LIN {X 0,Y 485.408,Z 513.857,A -85,B 0,C 180,E1 -6732.652,E2 -6732.652} C_VEL
LIN {X 0,Y 484.952,Z 527.725,A -85,B 0,C 180,E1 -6733.189,E2 -6733.189} C_VEL
LIN {X 0,Y 484.519,Z 541.1,A -85,B 0,C 180,E1 -6733.893,E2 -6733.893} C_VEL
LIN {X 0,Y 483.878,Z 553.705,A -85,B 0,C 180,E1 -6734.736,E2 -6734.736} C_VEL
LIN {X 0,Y 483.305,Z 565.203,A -85,B 0,C 180,E1 -6735.687,E2 -6735.687} C_VEL
LIN {X 0,Y 482.695,Z 575.753,A -85,B 0,C 180,E1 -6736.742,E2 -6736.742} C_VEL
LIN {X 0,Y 482.294,Z 585.397,A -85,B 0,C 180,E1 -6737.906,E2 -6737.906} C_VEL
LIN {X 0,Y 481.754,Z 594.848,A -85,B 0,C 180,E1 -6739.28,E2 -6739.28} C_VEL
LIN {X 0,Y 481.429,Z 602.033,A -85,B 0,C 180,E1 -6740.547,E2 -6740.547} C_VEL
LIN {X 0,Y 481.163,Z 608.903,A -85,B 0,C 180,E1 -6742.023,E2 -6742.023} C_VEL
LIN {X 0,Y 481.013,Z 614.317,A -85,B 0,C 180,E1 -6743.484,E2 -6743.484} C_VEL
LIN {X 0,Y 480.898,Z 618.563,A -85,B 0,C 180,E1 -6744.968,E2 -6744.968} C_VEL
LIN {X 0,Y 480.881,Z 621.983,A -85,B 0,C 180,E1 -6746.648,E2 -6746.648} C_VEL
LIN {X 0,Y 480.789,Z 624.022,A -85,B 0,C 180,E1 -6748.324,E2 -6748.324} C_VEL
LIN {X 0,Y 480.742,Z 624.729,A -85,B 0,C 180,E1 -6749.999,E2 -6749.999} C_VEL
LIN {X 0,Y 480.787,Z 624.108,A -85,B 0,C 180,E1 -6751.674,E2 -6751.674} C_VEL
LIN {X 0,Y 480.88,Z 622.144,A -85,B 0,C 180,E1 -6753.35,E2 -6753.35} C_VEL
LIN {X 0,Y 480.897,Z 618.796,A -85,B 0,C 180,E1 -6755.029,E2 -6755.029} C_VEL
LIN {X 0,Y 481.01,Z 613.965,A -85,B 0,C 180,E1 -6756.711,E2 -6756.711} C_VEL
LIN {X 0,Y 481.226,Z 607.51,A -85,B 0,C 180,E1 -6758.397,E2 -6758.397} C_VEL
LIN {X 0,Y 481.56,Z 600.315,A -85,B 0,C 180,E1 -6759.873,E2 -6759.873} C_VEL
LIN {X 0,Y 481.997,Z 591.359,A -85,B 0,C 180,E1 -6761.351,E2 -6761.351} C_VEL
LIN {X 0,Y 482.364,Z 581.99,A -85,B 0,C 180,E1 -6762.623,E2 -6762.623} C_VEL
LIN {X 0,Y 482.997,Z 571.618,A -85,B 0,C 180,E1 -6763.783,E2 -6763.783} C_VEL
LIN {X 0,Y 483.532,Z 560.185,A -85,B 0,C 180,E1 -6764.842,E2 -6764.842} C_VEL
LIN {X 0,Y 484.194,Z 547.528,A -85,B 0,C 180,E1 -6765.791,E2 -6765.791} C_VEL
LIN {X 0,Y 484.698,Z 535.279,A -85,B 0,C 180,E1 -6766.525,E2 -6766.525} C_VEL
LIN {X 0,Y 485.175,Z 521.511,A -85,B 0,C 180,E1 -6767.164,E2 -6767.164} C_VEL
LIN {X 0,Y 485.319,Z 512.158,A -85,B 0,C 180,E1 -6767.495,E2 -6767.495} C_VEL
LIN {X 0,Y 482.342,Z 497.804,A -85,B 0,C 180,E1 -6767.979,E2 -6767.979} C_VEL
LIN {X 0,Y 481.294,Z 492.955,A -85,B 0,C 180,E1 -6768.131,E2 -6768.131} C_VEL
LIN {X 0,Y 481.45,Z 484.218,A -85,B 0,C 180,E1 -6771.402,E2 -6771.402} C_VEL
LIN {X 0,Y 481.577,Z 476.033,A -85,B 0,C 180,E1 -6774.576,E2 -6774.576} C_VEL
LIN {X 0,Y 481.728,Z 467.861,A -85,B 0,C 180,E1 -6777.829,E2 -6777.829} C_VEL
LIN {X 0,Y 481.835,Z 460.745,A -85,B 0,C 180,E1 -6780.696,E2 -6780.696} C_VEL
LIN {X 0,Y 481.957,Z 453.069,A -85,B 0,C 180,E1 -6783.779,E2 -6783.779} C_VEL
LIN {X 0,Y 482.117,Z 445.735,A -85,B 0,C 180,E1 -6786.702,E2 -6786.702} C_VEL
LIN {X 0,Y 481.949,Z 440.341,A -85,B 0,C 180,E1 -6788.831,E2 -6788.831} C_VEL
LIN {X 0,Y 481.791,Z 439.1,A -85,B 0,C 180,E1 -6789.365,E2 -6789.365} C_VEL
LIN {X 0,Y 481.683,Z 439.11,A -85,B 0,C 180,E1 -6793.153,E2 -6793.153} C_VEL
LIN {X 0,Y 481.682,Z 439.11,A -85,B 0,C 180,E1 -6796.845,E2 -6796.845} C_VEL
LIN {X 0,Y 481.682,Z 439.108,A -85,B 0,C 180,E1 -6800.06,E2 -6800.06} C_VEL
LIN {X 0,Y 481.622,Z 439.12,A -85,B 0,C 180,E1 -6803.253,E2 -6803.253} C_VEL
LIN {X 0,Y 481.701,Z 439.107,A -85,B 0,C 180,E1 -6806.329,E2 -6806.329} C_VEL
LIN {X 0,Y 481.65,Z 439.109,A -85,B 0,C 180,E1 -6809.415,E2 -6809.415} C_VEL
LIN {X 0,Y 481.693,Z 439.106,A -85,B 0,C 180,E1 -6812.167,E2 -6812.167} C_VEL
LIN {X 0,Y 481.71,Z 439.106,A -85,B 0,C 180,E1 -6814.969,E2 -6814.969} C_VEL
LIN {X 0,Y 481.65,Z 439.106,A -85,B 0,C 180,E1 -6817.705,E2 -6817.705} C_VEL
LIN {X 0,Y 481.698,Z 439.111,A -85,B 0,C 180,E1 -6820.393,E2 -6820.393} C_VEL
LIN {X 0,Y 481.682,Z 439.107,A -85,B 0,C 180,E1 -6823.034,E2 -6823.034} C_VEL
LIN {X 0,Y 481.68,Z 439.112,A -85,B 0,C 180,E1 -6825.638,E2 -6825.638} C_VEL
LIN {X 0,Y 481.786,Z 439.092,A -85,B 0,C 180,E1 -6828.216,E2 -6828.216} C_VEL
LIN {X 0,Y 481.754,Z 439.096,A -85,B 0,C 180,E1 -6831.611,E2 -6831.611} C_VEL
LIN {X 0,Y 481.821,Z 439.095,A -85,B 0,C 180,E1 -6834.14,E2 -6834.14} C_VEL
LIN {X 0,Y 481.919,Z 439.082,A -85,B 0,C 180,E1 -6837.492,E2 -6837.492} C_VEL
LIN {X 0,Y 481.93,Z 439.077,A -85,B 0,C 180,E1 -6840,E2 -6840} C_VEL
LIN {X 0,Y 481.919,Z 439.077,A -85,B 0,C 180,E1 -6842.507,E2 -6842.507} C_VEL
LIN {X 0,Y 481.807,Z 439.09,A -85,B 0,C 180,E1 -6845.86,E2 -6845.86} C_VEL
LIN {X 0,Y 481.754,Z 439.099,A -85,B 0,C 180,E1 -6848.388,E2 -6848.388} C_VEL
LIN {X 0,Y 481.785,Z 439.094,A -85,B 0,C 180,E1 -6851.784,E2 -6851.784} C_VEL
LIN {X 0,Y 481.731,Z 439.102,A -85,B 0,C 180,E1 -6855.225,E2 -6855.225} C_VEL
LIN {X 0,Y 481.702,Z 439.107,A -85,B 0,C 180,E1 -6858.722,E2 -6858.722} C_VEL
LIN {X 0,Y 481.639,Z 439.113,A -85,B 0,C 180,E1 -6861.395,E2 -6861.395} C_VEL
LIN {X 0,Y 481.668,Z 439.111,A -85,B 0,C 180,E1 -6864.114,E2 -6864.114} C_VEL
LIN {X 0,Y 481.742,Z 439.106,A -85,B 0,C 180,E1 -6867.141,E2 -6867.141} C_VEL
LIN {X 0,Y 481.679,Z 439.108,A -85,B 0,C 180,E1 -6869.741,E2 -6869.741} C_VEL
LIN {X 0,Y 481.664,Z 439.112,A -85,B 0,C 180,E1 -6872.675,E2 -6872.675} C_VEL
LIN {X 0,Y 481.634,Z 439.119,A -85,B 0,C 180,E1 -6875.71,E2 -6875.71} C_VEL
LIN {X 0,Y 481.712,Z 439.109,A -85,B 0,C 180,E1 -6879.356,E2 -6879.356} C_VEL
LIN {X 0,Y 481.668,Z 439.11,A -85,B 0,C 180,E1 -6882.159,E2 -6882.159} C_VEL
LIN {X 0,Y 481.653,Z 439.117,A -85,B 0,C 180,E1 -6884.458,E2 -6884.458} C_VEL
LIN {X 0,Y 481.642,Z 439.118,A -85,B 0,C 180,E1 -6887.841,E2 -6887.841} C_VEL
LIN {X 0,Y 481.714,Z 439.105,A -85,B 0,C 180,E1 -6890.646,E2 -6890.646} C_VEL
LIN {X 0,Y 481.648,Z 439.16,A -85,B 0,C 180,E1 -6893.061,E2 -6893.061} C_VEL
LIN {X 0,Y 483.316,Z 447.33,A -85,B 0,C 180,E1 -6895.981,E2 -6895.981} C_VEL
LIN {X 0,Y 483.83,Z 451.8,A -85,B 0,C 180,E1 -6897.491,E2 -6897.491} C_VEL
LIN {X 0,Y 483.328,Z 460.852,A -85,B 0,C 180,E1 -6900.372,E2 -6900.372} C_VEL
LIN {X 0,Y 482.78,Z 471.48,A -85,B 0,C 180,E1 -6903.642,E2 -6903.642} C_VEL
LIN {X 0,Y 482.281,Z 482.192,A -85,B 0,C 180,E1 -6906.832,E2 -6906.832} C_VEL
LIN {X 0,Y 481.884,Z 492.95,A -85,B 0,C 180,E1 -6909.958,E2 -6909.958} C_VEL
LIN {X 0,Y 481.681,Z 500.305,A -85,B 0,C 180,E1 -6912.059,E2 -6912.059} C_VEL
LIN {X 0,Y 484.643,Z 516.718,A -85,B 0,C 180,E1 -6912.541,E2 -6912.541} C_VEL
LIN {X 0,Y 485.127,Z 520.38,A -85,B 0,C 180,E1 -6912.671,E2 -6912.671} C_VEL
LIN {X 0,Y 484.7,Z 534.321,A -85,B 0,C 180,E1 -6913.197,E2 -6913.197} C_VEL
LIN {X 0,Y 484.155,Z 547.998,A -85,B 0,C 180,E1 -6913.897,E2 -6913.897} C_VEL
LIN {X 0,Y 483.596,Z 560.749,A -85,B 0,C 180,E1 -6914.729,E2 -6914.729} C_VEL
LIN {X 0,Y 482.932,Z 573.657,A -85,B 0,C 180,E1 -6915.785,E2 -6915.785} C_VEL
LIN {X 0,Y 482.38,Z 585.261,A -85,B 0,C 180,E1 -6916.95,E2 -6916.95} C_VEL
LIN {X 0,Y 482.06,Z 593.893,A -85,B 0,C 180,E1 -6918.001,E2 -6918.001} C_VEL
LIN {X 0,Y 481.616,Z 602.799,A -85,B 0,C 180,E1 -6919.279,E2 -6919.279} C_VEL
LIN {X 0,Y 481.303,Z 611.222,A -85,B 0,C 180,E1 -6920.758,E2 -6920.758} C_VEL
LIN {X 0,Y 481.081,Z 617.116,A -85,B 0,C 180,E1 -6922.024,E2 -6922.024} C_VEL
LIN {X 0,Y 480.998,Z 622.715,A -85,B 0,C 180,E1 -6923.498,E2 -6923.498} C_VEL
LIN {X 0,Y 480.896,Z 626.971,A -85,B 0,C 180,E1 -6924.971,E2 -6924.971} C_VEL
LIN {X 0,Y 480.879,Z 630.438,A -85,B 0,C 180,E1 -6926.65,E2 -6926.65} C_VEL
LIN {X 0,Y 480.818,Z 632.466,A -85,B 0,C 180,E1 -6928.326,E2 -6928.326} C_VEL
LIN {X 0,Y 480.741,Z 633.146,A -85,B 0,C 180,E1 -6930.001,E2 -6930.001} C_VEL
LIN {X 0,Y 480.818,Z 632.438,A -85,B 0,C 180,E1 -6931.676,E2 -6931.676} C_VEL
LIN {X 0,Y 480.88,Z 630.341,A -85,B 0,C 180,E1 -6933.352,E2 -6933.352} C_VEL
LIN {X 0,Y 480.896,Z 626.844,A -85,B 0,C 180,E1 -6935.032,E2 -6935.032} C_VEL
LIN {X 0,Y 480.961,Z 622.613,A -85,B 0,C 180,E1 -6936.463,E2 -6936.463} C_VEL
LIN {X 0,Y 481.083,Z 616.893,A -85,B 0,C 180,E1 -6937.978,E2 -6937.978} C_VEL
LIN {X 0,Y 481.354,Z 609.746,A -85,B 0,C 180,E1 -6939.455,E2 -6939.455} C_VEL
LIN {X 0,Y 481.6,Z 602.307,A -85,B 0,C 180,E1 -6940.724,E2 -6940.724} C_VEL
LIN {X 0,Y 482.023,Z 593.342,A -85,B 0,C 180,E1 -6942.002,E2 -6942.002} C_VEL
LIN {X 0,Y 482.434,Z 582.489,A -85,B 0,C 180,E1 -6943.265,E2 -6943.265} C_VEL
LIN {X 0,Y 482.976,Z 570.326,A -85,B 0,C 180,E1 -6944.431,E2 -6944.431} C_VEL
LIN {X 0,Y 483.52,Z 559.588,A -85,B 0,C 180,E1 -6945.276,E2 -6945.276} C_VEL
LIN {X 0,Y 484.03,Z 546.618,A -85,B 0,C 180,E1 -6946.104,E2 -6946.104} C_VEL
LIN {X 0,Y 484.541,Z 532.544,A -85,B 0,C 180,E1 -6946.805,E2 -6946.805} C_VEL
LIN {X 0,Y 484.894,Z 518.9,A -85,B 0,C 180,E1 -6947.307,E2 -6947.307} C_VEL
LIN {X 0,Y 482.678,Z 505.977,A -85,B 0,C 180,E1 -6947.723,E2 -6947.723} C_VEL
LIN {X 0,Y 481.63,Z 499.829,A -85,B 0,C 180,E1 -6947.888,E2 -6947.888} C_VEL
LIN {X 0,Y 481.921,Z 488.783,A -85,B 0,C 180,E1 -6951.04,E2 -6951.04} C_VEL
LIN {X 0,Y 482.338,Z 478.56,A -85,B 0,C 180,E1 -6954.079,E2 -6954.079} C_VEL
LIN {X 0,Y 482.981,Z 468.006,A -85,B 0,C 180,E1 -6957.423,E2 -6957.423} C_VEL
LIN {X 0,Y 483.732,Z 458.94,A -85,B 0,C 180,E1 -6960.565,E2 -6960.565} C_VEL
LIN {X 0,Y 484.27,Z 453.447,A -85,B 0,C 180,E1 -6962.677,E2 -6962.677} C_VEL
LIN {X 0,Y 483.917,Z 450.215,A -85,B 0,C 180,E1 -6964.125,E2 -6964.125} C_VEL
LIN {X 0,Y 482.908,Z 445.184,A -85,B 0,C 180,E1 -6966.828,E2 -6966.828} C_VEL
LIN {X 0,Y 482.188,Z 441.559,A -85,B 0,C 180,E1 -6969.422,E2 -6969.422} C_VEL
LIN {X 0,Y 481.698,Z 439.328,A -85,B 0,C 180,E1 -6971.919,E2 -6971.919} C_VEL
LIN {X 0,Y 481.664,Z 439.115,A -85,B 0,C 180,E1 -6974.458,E2 -6974.458} C_VEL
LIN {X 0,Y 481.659,Z 439.116,A -85,B 0,C 180,E1 -6977.84,E2 -6977.84} C_VEL
LIN {X 0,Y 481.935,Z 440.548,A -85,B 0,C 180,E1 -6980.085,E2 -6980.085} C_VEL
LIN {X 0,Y 482.31,Z 442.658,A -85,B 0,C 180,E1 -6982.265,E2 -6982.265} C_VEL
LIN {X 0,Y 482.566,Z 445.208,A -85,B 0,C 180,E1 -6984.37,E2 -6984.37} C_VEL
LIN {X 0,Y 482.395,Z 448.059,A -85,B 0,C 180,E1 -6986.384,E2 -6986.384} C_VEL
LIN {X 0,Y 482.07,Z 452.653,A -85,B 0,C 180,E1 -6989.334,E2 -6989.334} C_VEL
LIN {X 0,Y 481.831,Z 457.403,A -85,B 0,C 180,E1 -6992.176,E2 -6992.176} C_VEL
LIN {X 0,Y 481.632,Z 462.281,A -85,B 0,C 180,E1 -6994.965,E2 -6994.965} C_VEL
LIN {X 0,Y 481.481,Z 467.233,A -85,B 0,C 180,E1 -6997.697,E2 -6997.697} C_VEL
LIN {X 0,Y 481.309,Z 472.23,A -85,B 0,C 180,E1 -7000.376,E2 -7000.376} C_VEL
LIN {X 0,Y 481.179,Z 477.249,A -85,B 0,C 180,E1 -7003.015,E2 -7003.015} C_VEL
LIN {X 0,Y 481.177,Z 481.115,A -85,B 0,C 180,E1 -7004.991,E2 -7004.991} C_VEL
LIN {X 0,Y 483.851,Z 494.163,A -85,B 0,C 180,E1 -7005.476,E2 -7005.476} C_VEL
LIN {X 0,Y 484.115,Z 498.642,A -85,B 0,C 180,E1 -7005.659,E2 -7005.659} C_VEL
LIN {X 0,Y 483.737,Z 510.946,A -85,B 0,C 180,E1 -7006.237,E2 -7006.237} C_VEL
LIN {X 0,Y 483.337,Z 522.757,A -85,B 0,C 180,E1 -7006.964,E2 -7006.964} C_VEL
LIN {X 0,Y 482.919,Z 533.788,A -85,B 0,C 180,E1 -7007.818,E2 -7007.818} C_VEL
LIN {X 0,Y 482.46,Z 542.691,A -85,B 0,C 180,E1 -7008.659,E2 -7008.659} C_VEL
LIN {X 0,Y 482.05,Z 551.892,A -85,B 0,C 180,E1 -7009.712,E2 -7009.712} C_VEL
LIN {X 0,Y 481.693,Z 560.831,A -85,B 0,C 180,E1 -7010.976,E2 -7010.976} C_VEL
LIN {X 0,Y 481.367,Z 568.059,A -85,B 0,C 180,E1 -7012.238,E2 -7012.238} C_VEL
LIN {X 0,Y 481.191,Z 574.235,A -85,B 0,C 180,E1 -7013.601,E2 -7013.601} C_VEL
LIN {X 0,Y 480.918,Z 579.013,A -85,B 0,C 180,E1 -7014.97,E2 -7014.97} C_VEL
LIN {X 0,Y 481.043,Z 581.302,A -85,B 0,C 180,E1 -7015.811,E2 -7015.811} C_VEL
LIN {X 0,Y 480.913,Z 583.174,A -85,B 0,C 180,E1 -7016.649,E2 -7016.649} C_VEL
LIN {X 0,Y 480.927,Z 584.583,A -85,B 0,C 180,E1 -7017.487,E2 -7017.487} C_VEL
LIN {X 0,Y 480.761,Z 586.185,A -85,B 0,C 180,E1 -7019.162,E2 -7019.162} C_VEL
LIN {X 0,Y 480.743,Z 586.404,A -85,B 0,C 180,E1 -7020,E2 -7020} C_VEL
LIN {X 0,Y 480.761,Z 586.199,A -85,B 0,C 180,E1 -7020.838,E2 -7020.838} C_VEL
LIN {X 0,Y 480.911,Z 584.58,A -85,B 0,C 180,E1 -7022.513,E2 -7022.513} C_VEL
LIN {X 0,Y 480.913,Z 583.184,A -85,B 0,C 180,E1 -7023.351,E2 -7023.351} C_VEL
LIN {X 0,Y 480.979,Z 580.252,A -85,B 0,C 180,E1 -7024.61,E2 -7024.61} C_VEL
LIN {X 0,Y 481.128,Z 576.286,A -85,B 0,C 180,E1 -7025.869,E2 -7025.869} C_VEL
LIN {X 0,Y 481.198,Z 571.186,A -85,B 0,C 180,E1 -7027.131,E2 -7027.131} C_VEL
LIN {X 0,Y 481.468,Z 564.77,A -85,B 0,C 180,E1 -7028.394,E2 -7028.394} C_VEL
LIN {X 0,Y 481.762,Z 556.769,A -85,B 0,C 180,E1 -7029.658,E2 -7029.658} C_VEL
LIN {X 0,Y 482.102,Z 548.627,A -85,B 0,C 180,E1 -7030.712,E2 -7030.712} C_VEL
LIN {X 0,Y 482.591,Z 538.728,A -85,B 0,C 180,E1 -7031.764,E2 -7031.764} C_VEL
LIN {X 0,Y 483.002,Z 529.038,A -85,B 0,C 180,E1 -7032.607,E2 -7032.607} C_VEL
LIN {X 0,Y 483.398,Z 516.896,A -85,B 0,C 180,E1 -7033.451,E2 -7033.451} C_VEL
LIN {X 0,Y 483.857,Z 504.112,A -85,B 0,C 180,E1 -7034.135,E2 -7034.135} C_VEL
LIN {X 0,Y 483.912,Z 495.387,A -85,B 0,C 180,E1 -7034.495,E2 -7034.495} C_VEL
LIN {X 0,Y 481.647,Z 483.267,A -85,B 0,C 180,E1 -7034.946,E2 -7034.946} C_VEL
LIN {X 0,Y 481.064,Z 480.208,A -85,B 0,C 180,E1 -7035.057,E2 -7035.057} C_VEL
LIN {X 0,Y 481.163,Z 473.733,A -85,B 0,C 180,E1 -7038.301,E2 -7038.301} C_VEL
LIN {X 0,Y 481.246,Z 467.64,A -85,B 0,C 180,E1 -7041.413,E2 -7041.413} C_VEL
LIN {X 0,Y 481.364,Z 462.394,A -85,B 0,C 180,E1 -7044.13,E2 -7044.13} C_VEL
LIN {X 0,Y 481.499,Z 456.791,A -85,B 0,C 180,E1 -7047.08,E2 -7047.08} C_VEL
LIN {X 0,Y 481.631,Z 451.796,A -85,B 0,C 180,E1 -7049.744,E2 -7049.744} C_VEL
LIN {X 0,Y 481.742,Z 446.423,A -85,B 0,C 180,E1 -7052.669,E2 -7052.669} C_VEL
LIN {X 0,Y 481.877,Z 441.781,A -85,B 0,C 180,E1 -7055.239,E2 -7055.239} C_VEL
LIN {X 0,Y 481.697,Z 439.111,A -85,B 0,C 180,E1 -7056.871,E2 -7056.871} C_VEL
LIN {X 0,Y 481.682,Z 439.11,A -85,B 0,C 180,E1 -7059.94,E2 -7059.94} C_VEL
LIN {X 0,Y 481.672,Z 439.113,A -85,B 0,C 180,E1 -7063.296,E2 -7063.296} C_VEL
LIN {X 0,Y 481.664,Z 439.115,A -85,B 0,C 180,E1 -7065.64,E2 -7065.64} C_VEL
LIN {X 0,Y 481.67,Z 439.115,A -85,B 0,C 180,E1 -7068.959,E2 -7068.959} C_VEL
LIN {X 0,Y 481.772,Z 439.213,A -85,B 0,C 180,E1 -7070.807,E2 -7070.807} C_VEL
LIN {X 0,Y 482.15,Z 444.175,A -85,B 0,C 180,E1 -7072.776,E2 -7072.776} C_VEL
LIN {X 0,Y 481.992,Z 451.806,A -85,B 0,C 180,E1 -7075.825,E2 -7075.825} C_VEL
LIN {X 0,Y 481.866,Z 459.266,A -85,B 0,C 180,E1 -7078.817,E2 -7078.817} C_VEL
LIN {X 0,Y 481.723,Z 466.755,A -85,B 0,C 180,E1 -7081.829,E2 -7081.829} C_VEL
LIN {X 0,Y 481.046,Z 468.496,A -85,B 0,C 180,E1 -7082.495,E2 -7082.495} C_VEL
LIN {X 0,Y 478.153,Z 471.535,A -85,B 0,C 180,E1 -7083.569,E2 -7083.569} C_VEL
LIN {X 0,Y 475.691,Z 473.992,A -85,B 0,C 180,E1 -7084.433,E2 -7084.433} C_VEL
LIN {X 0,Y 474.611,Z 475.8,A -85,B 0,C 180,E1 -7085.104,E2 -7085.104} C_VEL
LIN {X 0,Y 474.51,Z 476.385,A -85,B 0,C 180,E1 -7085.332,E2 -7085.332} C_VEL
LIN {X 0,Y 474.403,Z 483.867,A -85,B 0,C 180,E1 -7088.261,E2 -7088.261} C_VEL
LIN {X 0,Y 474.273,Z 491.025,A -85,B 0,C 180,E1 -7090.972,E2 -7090.972} C_VEL
LIN {X 0,Y 474.257,Z 492.969,A -85,B 0,C 180,E1 -7091.7,E2 -7091.7} C_VEL
LIN {X 0,Y 477.7,Z 508.75,A -85,B 0,C 180,E1 -7092.197,E2 -7092.197} C_VEL
LIN {X 0,Y 478.636,Z 514.739,A -85,B 0,C 180,E1 -7092.426,E2 -7092.426} C_VEL
LIN {X 0,Y 478.137,Z 528.619,A -85,B 0,C 180,E1 -7092.984,E2 -7092.984} C_VEL
LIN {X 0,Y 477.674,Z 541.222,A -85,B 0,C 180,E1 -7093.661,E2 -7093.661} C_VEL
LIN {X 0,Y 477.022,Z 553.755,A -85,B 0,C 180,E1 -7094.511,E2 -7094.511} C_VEL
LIN {X 0,Y 476.485,Z 564.109,A -85,B 0,C 180,E1 -7095.368,E2 -7095.368} C_VEL
LIN {X 0,Y 475.905,Z 573.893,A -85,B 0,C 180,E1 -7096.332,E2 -7096.332} C_VEL
LIN {X 0,Y 475.294,Z 584.235,A -85,B 0,C 180,E1 -7097.56,E2 -7097.56} C_VEL
LIN {X 0,Y 474.866,Z 593.572,A -85,B 0,C 180,E1 -7098.906,E2 -7098.906} C_VEL
LIN {X 0,Y 474.409,Z 602.087,A -85,B 0,C 180,E1 -7100.405,E2 -7100.405} C_VEL
LIN {X 0,Y 474.124,Z 608.958,A -85,B 0,C 180,E1 -7101.904,E2 -7101.904} C_VEL
LIN {X 0,Y 473.937,Z 614.699,A -85,B 0,C 180,E1 -7103.486,E2 -7103.486} C_VEL
LIN {X 0,Y 473.835,Z 618.619,A -85,B 0,C 180,E1 -7104.893,E2 -7104.893} C_VEL
LIN {X 0,Y 473.789,Z 622.039,A -85,B 0,C 180,E1 -7106.597,E2 -7106.597} C_VEL
LIN {X 0,Y 473.694,Z 624.078,A -85,B 0,C 180,E1 -7108.299,E2 -7108.299} C_VEL
LIN {X 0,Y 473.668,Z 624.785,A -85,B 0,C 180,E1 -7109.999,E2 -7109.999} C_VEL
LIN {X 0,Y 473.692,Z 624.163,A -85,B 0,C 180,E1 -7111.699,E2 -7111.699} C_VEL
LIN {X 0,Y 473.788,Z 622.198,A -85,B 0,C 180,E1 -7113.401,E2 -7113.401} C_VEL
LIN {X 0,Y 473.834,Z 618.848,A -85,B 0,C 180,E1 -7115.105,E2 -7115.105} C_VEL
LIN {X 0,Y 473.926,Z 614.016,A -85,B 0,C 180,E1 -7116.812,E2 -7116.812} C_VEL
LIN {X 0,Y 474.161,Z 607.559,A -85,B 0,C 180,E1 -7118.523,E2 -7118.523} C_VEL
LIN {X 0,Y 474.52,Z 600.363,A -85,B 0,C 180,E1 -7120.021,E2 -7120.021} C_VEL
LIN {X 0,Y 474.998,Z 591.404,A -85,B 0,C 180,E1 -7121.521,E2 -7121.521} C_VEL
LIN {X 0,Y 475.393,Z 582.032,A -85,B 0,C 180,E1 -7122.811,E2 -7122.811} C_VEL
LIN {X 0,Y 476.071,Z 571.658,A -85,B 0,C 180,E1 -7123.988,E2 -7123.988} C_VEL
LIN {X 0,Y 476.65,Z 560.221,A -85,B 0,C 180,E1 -7125.061,E2 -7125.061} C_VEL
LIN {X 0,Y 477.36,Z 547.557,A -85,B 0,C 180,E1 -7126.023,E2 -7126.023} C_VEL
LIN {X 0,Y 477.954,Z 534.001,A -85,B 0,C 180,E1 -7126.838,E2 -7126.838} C_VEL
LIN {X 0,Y 478.42,Z 519.79,A -85,B 0,C 180,E1 -7127.481,E2 -7127.481} C_VEL
LIN {X 0,Y 478.588,Z 513.604,A -85,B 0,C 180,E1 -7127.702,E2 -7127.702} C_VEL
LIN {X 0,Y 475.787,Z 499.927,A -85,B 0,C 180,E1 -7128.189,E2 -7128.189} C_VEL
LIN {X 0,Y 474.275,Z 492.985,A -85,B 0,C 180,E1 -7128.387,E2 -7128.387} C_VEL
LIN {X 0,Y 474.41,Z 484.115,A -85,B 0,C 180,E1 -7131.736,E2 -7131.736} C_VEL
LIN {X 0,Y 474.549,Z 475.931,A -85,B 0,C 180,E1 -7134.942,E2 -7134.942} C_VEL
LIN {X 0,Y 474.696,Z 467.635,A -85,B 0,C 180,E1 -7138.278,E2 -7138.278} C_VEL
LIN {X 0,Y 474.826,Z 460.456,A -85,B 0,C 180,E1 -7141.199,E2 -7141.199} C_VEL
LIN {X 0,Y 474.962,Z 451.758,A -85,B 0,C 180,E1 -7144.726,E2 -7144.726} C_VEL
LIN {X 0,Y 475.13,Z 443.992,A -85,B 0,C 180,E1 -7147.842,E2 -7147.842} C_VEL
LIN {X 0,Y 474.724,Z 439.98,A -85,B 0,C 180,E1 -7149.536,E2 -7149.536} C_VEL
LIN {X 0,Y 474.646,Z 439.989,A -85,B 0,C 180,E1 -7152.929,E2 -7152.929} C_VEL
LIN {X 0,Y 474.612,Z 439.994,A -85,B 0,C 180,E1 -7155.895,E2 -7155.895} C_VEL
LIN {X 0,Y 474.639,Z 439.988,A -85,B 0,C 180,E1 -7159.037,E2 -7159.037} C_VEL
LIN {X 0,Y 474.609,Z 439.99,A -85,B 0,C 180,E1 -7161.702,E2 -7161.702} C_VEL
LIN {X 0,Y 474.622,Z 439.991,A -85,B 0,C 180,E1 -7164.725,E2 -7164.725} C_VEL
LIN {X 0,Y 474.629,Z 439.989,A -85,B 0,C 180,E1 -7167.787,E2 -7167.787} C_VEL
LIN {X 0,Y 474.623,Z 439.988,A -85,B 0,C 180,E1 -7170.882,E2 -7170.882} C_VEL
LIN {X 0,Y 474.657,Z 439.983,A -85,B 0,C 180,E1 -7173.628,E2 -7173.628} C_VEL
LIN {X 0,Y 474.626,Z 439.99,A -85,B 0,C 180,E1 -7176.64,E2 -7176.64} C_VEL
LIN {X 0,Y 474.666,Z 439.981,A -85,B 0,C 180,E1 -7179.185,E2 -7179.185} C_VEL
LIN {X 0,Y 474.647,Z 439.987,A -85,B 0,C 180,E1 -7181.884,E2 -7181.884} C_VEL
LIN {X 0,Y 474.689,Z 439.978,A -85,B 0,C 180,E1 -7184.544,E2 -7184.544} C_VEL
LIN {X 0,Y 474.729,Z 439.971,A -85,B 0,C 180,E1 -7188.038,E2 -7188.038} C_VEL
LIN {X 0,Y 474.719,Z 439.973,A -85,B 0,C 180,E1 -7191.486,E2 -7191.486} C_VEL
LIN {X 0,Y 474.781,Z 439.971,A -85,B 0,C 180,E1 -7194.052,E2 -7194.052} C_VEL
LIN {X 0,Y 474.886,Z 439.958,A -85,B 0,C 180,E1 -7197.455,E2 -7197.455} C_VEL
LIN {X 0,Y 474.867,Z 439.959,A -85,B 0,C 180,E1 -7200.848,E2 -7200.848} C_VEL
LIN {X 0,Y 474.885,Z 439.953,A -85,B 0,C 180,E1 -7202.545,E2 -7202.545} C_VEL
LIN {X 0,Y 474.77,Z 439.967,A -85,B 0,C 180,E1 -7205.948,E2 -7205.948} C_VEL
LIN {X 0,Y 474.719,Z 439.974,A -85,B 0,C 180,E1 -7208.514,E2 -7208.514} C_VEL
LIN {X 0,Y 474.728,Z 439.973,A -85,B 0,C 180,E1 -7211.962,E2 -7211.962} C_VEL
LIN {X 0,Y 474.67,Z 439.978,A -85,B 0,C 180,E1 -7215.768,E2 -7215.768} C_VEL
LIN {X 0,Y 474.655,Z 439.982,A -85,B 0,C 180,E1 -7219.011,E2 -7219.011} C_VEL
LIN {X 0,Y 474.583,Z 439.995,A -85,B 0,C 180,E1 -7221.729,E2 -7221.729} C_VEL
LIN {X 0,Y 474.649,Z 439.983,A -85,B 0,C 180,E1 -7224.493,E2 -7224.493} C_VEL
LIN {X 0,Y 474.689,Z 439.981,A -85,B 0,C 180,E1 -7227.339,E2 -7227.339} C_VEL
LIN {X 0,Y 474.601,Z 439.993,A -85,B 0,C 180,E1 -7230.812,E2 -7230.812} C_VEL
LIN {X 0,Y 474.629,Z 439.99,A -85,B 0,C 180,E1 -7233.985,E2 -7233.985} C_VEL
LIN {X 0,Y 474.567,Z 439.993,A -85,B 0,C 180,E1 -7236.901,E2 -7236.901} C_VEL
LIN {X 0,Y 474.647,Z 439.986,A -85,B 0,C 180,E1 -7239.653,E2 -7239.653} C_VEL
LIN {X 0,Y 474.645,Z 439.989,A -85,B 0,C 180,E1 -7242.931,E2 -7242.931} C_VEL
LIN {X 0,Y 474.602,Z 439.993,A -85,B 0,C 180,E1 -7245.896,E2 -7245.896} C_VEL
LIN {X 0,Y 474.634,Z 439.988,A -85,B 0,C 180,E1 -7249.04,E2 -7249.04} C_VEL
LIN {X 0,Y 474.614,Z 439.99,A -85,B 0,C 180,E1 -7251.704,E2 -7251.704} C_VEL
LIN {X 0,Y 474.628,Z 440.036,A -85,B 0,C 180,E1 -7252.757,E2 -7252.757} C_VEL
LIN {X 0,Y 476.347,Z 448.699,A -85,B 0,C 180,E1 -7255.901,E2 -7255.901} C_VEL
LIN {X 0,Y 476.841,Z 452.3,A -85,B 0,C 180,E1 -7257.151,E2 -7257.151} C_VEL
LIN {X 0,Y 476.518,Z 459.264,A -85,B 0,C 180,E1 -7259.416,E2 -7259.416} C_VEL
LIN {X 0,Y 475.963,Z 468.62,A -85,B 0,C 180,E1 -7262.369,E2 -7262.369} C_VEL
LIN {X 0,Y 475.494,Z 477.461,A -85,B 0,C 180,E1 -7265.088,E2 -7265.088} C_VEL
LIN {X 0,Y 475.046,Z 488.172,A -85,B 0,C 180,E1 -7268.294,E2 -7268.294} C_VEL
LIN {X 0,Y 474.651,Z 499.486,A -85,B 0,C 180,E1 -7271.601,E2 -7271.601} C_VEL
LIN {X 0,Y 474.668,Z 500.219,A -85,B 0,C 180,E1 -7271.815,E2 -7271.815} C_VEL
LIN {X 0,Y 477.433,Z 515.65,A -85,B 0,C 180,E1 -7272.267,E2 -7272.267} C_VEL
LIN {X 0,Y 478.258,Z 521.165,A -85,B 0,C 180,E1 -7272.469,E2 -7272.469} C_VEL
LIN {X 0,Y 477.806,Z 534.798,A -85,B 0,C 180,E1 -7273.005,E2 -7273.005} C_VEL
LIN {X 0,Y 477.226,Z 548.905,A -85,B 0,C 180,E1 -7273.752,E2 -7273.752} C_VEL
LIN {X 0,Y 476.592,Z 561.601,A -85,B 0,C 180,E1 -7274.608,E2 -7274.608} C_VEL
LIN {X 0,Y 475.921,Z 574.27,A -85,B 0,C 180,E1 -7275.681,E2 -7275.681} C_VEL
LIN {X 0,Y 475.4,Z 584.782,A -85,B 0,C 180,E1 -7276.755,E2 -7276.755} C_VEL
LIN {X 0,Y 475.016,Z 593.817,A -85,B 0,C 180,E1 -7277.873,E2 -7277.873} C_VEL
LIN {X 0,Y 474.595,Z 602.37,A -85,B 0,C 180,E1 -7279.118,E2 -7279.118} C_VEL
LIN {X 0,Y 474.244,Z 610.819,A -85,B 0,C 180,E1 -7280.619,E2 -7280.619} C_VEL
LIN {X 0,Y 473.998,Z 616.729,A -85,B 0,C 180,E1 -7281.904,E2 -7281.904} C_VEL
LIN {X 0,Y 473.917,Z 622.703,A -85,B 0,C 180,E1 -7283.506,E2 -7283.506} C_VEL
LIN {X 0,Y 473.829,Z 626.614,A -85,B 0,C 180,E1 -7284.895,E2 -7284.895} C_VEL
LIN {X 0,Y 473.727,Z 628.563,A -85,B 0,C 180,E1 -7285.747,E2 -7285.747} C_VEL
LIN {X 0,Y 473.805,Z 630.094,A -85,B 0,C 180,E1 -7286.6,E2 -7286.6} C_VEL
LIN {X 0,Y 473.75,Z 632.121,A -85,B 0,C 180,E1 -7288.301,E2 -7288.301} C_VEL
LIN {X 0,Y 473.668,Z 632.805,A -85,B 0,C 180,E1 -7290.001,E2 -7290.001} C_VEL
LIN {X 0,Y 473.75,Z 632.088,A -85,B 0,C 180,E1 -7291.701,E2 -7291.701} C_VEL
LIN {X 0,Y 473.806,Z 629.969,A -85,B 0,C 180,E1 -7293.403,E2 -7293.403} C_VEL
LIN {X 0,Y 473.829,Z 626.459,A -85,B 0,C 180,E1 -7295.107,E2 -7295.107} C_VEL
LIN {X 0,Y 473.869,Z 622.585,A -85,B 0,C 180,E1 -7296.442,E2 -7296.442} C_VEL
LIN {X 0,Y 473.999,Z 616.458,A -85,B 0,C 180,E1 -7298.098,E2 -7298.098} C_VEL
LIN {X 0,Y 474.274,Z 609.255,A -85,B 0,C 180,E1 -7299.597,E2 -7299.597} C_VEL
LIN {X 0,Y 474.583,Z 601.949,A -85,B 0,C 180,E1 -7300.884,E2 -7300.884} C_VEL
LIN {X 0,Y 475.034,Z 592.199,A -85,B 0,C 180,E1 -7302.298,E2 -7302.298} C_VEL
LIN {X 0,Y 475.495,Z 582.404,A -85,B 0,C 180,E1 -7303.462,E2 -7303.462} C_VEL
LIN {X 0,Y 476.03,Z 571.54,A -85,B 0,C 180,E1 -7304.537,E2 -7304.537} C_VEL
LIN {X 0,Y 476.647,Z 559.58,A -85,B 0,C 180,E1 -7305.501,E2 -7305.501} C_VEL
LIN {X 0,Y 477.206,Z 546.759,A -85,B 0,C 180,E1 -7306.33,E2 -7306.33} C_VEL
LIN {X 0,Y 477.668,Z 533.554,A -85,B 0,C 180,E1 -7306.99,E2 -7306.99} C_VEL
LIN {X 0,Y 478.006,Z 519.79,A -85,B 0,C 180,E1 -7307.505,E2 -7307.505} C_VEL
LIN {X 0,Y 475.677,Z 505.777,A -85,B 0,C 180,E1 -7307.973,E2 -7307.973} C_VEL
LIN {X 0,Y 474.595,Z 499.634,A -85,B 0,C 180,E1 -7308.153,E2 -7308.153} C_VEL
LIN {X 0,Y 474.898,Z 489.196,A -85,B 0,C 180,E1 -7311.198,E2 -7311.198} C_VEL
LIN {X 0,Y 475.314,Z 480.014,A -85,B 0,C 180,E1 -7313.993,E2 -7313.993} C_VEL
LIN {X 0,Y 475.939,Z 469.948,A -85,B 0,C 180,E1 -7317.244,E2 -7317.244} C_VEL
LIN {X 0,Y 476.773,Z 460.552,A -85,B 0,C 180,E1 -7320.569,E2 -7320.569} C_VEL
LIN {X 0,Y 477.377,Z 455.682,A -85,B 0,C 180,E1 -7322.472,E2 -7322.472} C_VEL
LIN {X 0,Y 477.1,Z 452.207,A -85,B 0,C 180,E1 -7324.04,E2 -7324.04} C_VEL
LIN {X 0,Y 476.287,Z 448.221,A -85,B 0,C 180,E1 -7326.174,E2 -7326.174} C_VEL
LIN {X 0,Y 475.621,Z 444.776,A -85,B 0,C 180,E1 -7328.45,E2 -7328.45} C_VEL
LIN {X 0,Y 475.087,Z 442.035,A -85,B 0,C 180,E1 -7331.023,E2 -7331.023} C_VEL
LIN {X 0,Y 474.705,Z 440.644,A -85,B 0,C 180,E1 -7333.494,E2 -7333.494} C_VEL
LIN {X 0,Y 474.682,Z 440.399,A -85,B 0,C 180,E1 -7335.904,E2 -7335.904} C_VEL
LIN {X 0,Y 474.851,Z 441.145,A -85,B 0,C 180,E1 -7338.239,E2 -7338.239} C_VEL
LIN {X 0,Y 475.152,Z 442.691,A -85,B 0,C 180,E1 -7340.505,E2 -7340.505} C_VEL
LIN {X 0,Y 475.527,Z 445.078,A -85,B 0,C 180,E1 -7342.949,E2 -7342.949} C_VEL
LIN {X 0,Y 475.625,Z 447.342,A -85,B 0,C 180,E1 -7344.811,E2 -7344.811} C_VEL
LIN {X 0,Y 475.238,Z 451.667,A -85,B 0,C 180,E1 -7347.834,E2 -7347.834} C_VEL
LIN {X 0,Y 474.961,Z 456.338,A -85,B 0,C 180,E1 -7350.813,E2 -7350.813} C_VEL
LIN {X 0,Y 474.699,Z 461.065,A -85,B 0,C 180,E1 -7353.631,E2 -7353.631} C_VEL
LIN {X 0,Y 474.517,Z 466.385,A -85,B 0,C 180,E1 -7356.676,E2 -7356.676} C_VEL
LIN {X 0,Y 474.363,Z 470.905,A -85,B 0,C 180,E1 -7359.171,E2 -7359.171} C_VEL
LIN {X 0,Y 474.22,Z 475.908,A -85,B 0,C 180,E1 -7361.867,E2 -7361.867} C_VEL
LIN {X 0,Y 474.112,Z 481.292,A -85,B 0,C 180,E1 -7364.708,E2 -7364.708} C_VEL
LIN {X 0,Y 476.882,Z 494.048,A -85,B 0,C 180,E1 -7365.218,E2 -7365.218} C_VEL
LIN {X 0,Y 477.292,Z 499.417,A -85,B 0,C 180,E1 -7365.449,E2 -7365.449} C_VEL
LIN {X 0,Y 476.874,Z 511.455,A -85,B 0,C 180,E1 -7366.035,E2 -7366.035} C_VEL
LIN {X 0,Y 476.421,Z 523.738,A -85,B 0,C 180,E1 -7366.81,E2 -7366.81} C_VEL
LIN {X 0,Y 475.948,Z 535.37,A -85,B 0,C 180,E1 -7367.745,E2 -7367.745} C_VEL
LIN {X 0,Y 475.455,Z 545.028,A -85,B 0,C 180,E1 -7368.705,E2 -7368.705} C_VEL
LIN {X 0,Y 474.995,Z 553.87,A -85,B 0,C 180,E1 -7369.773,E2 -7369.773} C_VEL
LIN {X 0,Y 474.625,Z 562.536,A -85,B 0,C 180,E1 -7371.055,E2 -7371.055} C_VEL
LIN {X 0,Y 474.287,Z 569.465,A -85,B 0,C 180,E1 -7372.336,E2 -7372.336} C_VEL
LIN {X 0,Y 474.142,Z 574.849,A -85,B 0,C 180,E1 -7373.576,E2 -7373.576} C_VEL
LIN {X 0,Y 473.858,Z 579.364,A -85,B 0,C 180,E1 -7374.895,E2 -7374.895} C_VEL
LIN {X 0,Y 473.982,Z 581.651,A -85,B 0,C 180,E1 -7375.748,E2 -7375.748} C_VEL
LIN {X 0,Y 473.848,Z 583.526,A -85,B 0,C 180,E1 -7376.599,E2 -7376.599} C_VEL
LIN {X 0,Y 473.837,Z 584.937,A -85,B 0,C 180,E1 -7377.45,E2 -7377.45} C_VEL
LIN {X 0,Y 473.69,Z 586.535,A -85,B 0,C 180,E1 -7379.15,E2 -7379.15} C_VEL
LIN {X 0,Y 473.67,Z 586.751,A -85,B 0,C 180,E1 -7380,E2 -7380} C_VEL
LIN {X 0,Y 473.689,Z 586.541,A -85,B 0,C 180,E1 -7380.85,E2 -7380.85} C_VEL
LIN {X 0,Y 473.761,Z 585.919,A -85,B 0,C 180,E1 -7381.7,E2 -7381.7} C_VEL
LIN {X 0,Y 473.822,Z 584.908,A -85,B 0,C 180,E1 -7382.55,E2 -7382.55} C_VEL
LIN {X 0,Y 473.849,Z 583.505,A -85,B 0,C 180,E1 -7383.401,E2 -7383.401} C_VEL
LIN {X 0,Y 473.902,Z 580.559,A -85,B 0,C 180,E1 -7384.679,E2 -7384.679} C_VEL
LIN {X 0,Y 474.071,Z 576.576,A -85,B 0,C 180,E1 -7385.957,E2 -7385.957} C_VEL
LIN {X 0,Y 474.151,Z 571.458,A -85,B 0,C 180,E1 -7387.238,E2 -7387.238} C_VEL
LIN {X 0,Y 474.434,Z 565.021,A -85,B 0,C 180,E1 -7388.519,E2 -7388.519} C_VEL
LIN {X 0,Y 474.751,Z 556.997,A -85,B 0,C 180,E1 -7389.802,E2 -7389.802} C_VEL
LIN {X 0,Y 475.127,Z 548.84,A -85,B 0,C 180,E1 -7390.871,E2 -7390.871} C_VEL
LIN {X 0,Y 475.655,Z 538.93,A -85,B 0,C 180,E1 -7391.938,E2 -7391.938} C_VEL
LIN {X 0,Y 476.117,Z 527.495,A -85,B 0,C 180,E1 -7392.928,E2 -7392.928} C_VEL
LIN {X 0,Y 476.586,Z 515.378,A -85,B 0,C 180,E1 -7393.756,E2 -7393.756} C_VEL
LIN {X 0,Y 477.018,Z 503.206,A -85,B 0,C 180,E1 -7394.396,E2 -7394.396} C_VEL
LIN {X 0,Y 477.016,Z 496.065,A -85,B 0,C 180,E1 -7394.696,E2 -7394.696} C_VEL
LIN {X 0,Y 474.703,Z 483.952,A -85,B 0,C 180,E1 -7395.164,E2 -7395.164} C_VEL
LIN {X 0,Y 473.973,Z 480.314,A -85,B 0,C 180,E1 -7395.303,E2 -7395.303} C_VEL
LIN {X 0,Y 474.099,Z 474.176,A -85,B 0,C 180,E1 -7398.425,E2 -7398.425} C_VEL
LIN {X 0,Y 474.185,Z 467.739,A -85,B 0,C 180,E1 -7401.748,E2 -7401.748} C_VEL
LIN {X 0,Y 474.309,Z 462.467,A -85,B 0,C 180,E1 -7404.512,E2 -7404.512} C_VEL
LIN {X 0,Y 474.462,Z 457.158,A -85,B 0,C 180,E1 -7407.335,E2 -7407.335} C_VEL
LIN {X 0,Y 474.591,Z 451.809,A -85,B 0,C 180,E1 -7410.231,E2 -7410.231} C_VEL
LIN {X 0,Y 474.757,Z 446.406,A -85,B 0,C 180,E1 -7413.211,E2 -7413.211} C_VEL
LIN {X 0,Y 474.85,Z 442.32,A -85,B 0,C 180,E1 -7415.508,E2 -7415.508} C_VEL
LIN {X 0,Y 474.645,Z 439.99,A -85,B 0,C 180,E1 -7416.91,E2 -7416.91} C_VEL
LIN {X 0,Y 474.633,Z 439.99,A -85,B 0,C 180,E1 -7419.647,E2 -7419.647} C_VEL
LIN {X 0,Y 474.641,Z 439.989,A -85,B 0,C 180,E1 -7422.932,E2 -7422.932} C_VEL
LIN {X 0,Y 474.615,Z 439.994,A -85,B 0,C 180,E1 -7425.895,E2 -7425.895} C_VEL
LIN {X 0,Y 474.644,Z 439.99,A -85,B 0,C 180,E1 -7429.039,E2 -7429.039} C_VEL
LIN {X 0,Y 474.722,Z 440.056,A -85,B 0,C 180,E1 -7430.667,E2 -7430.667} C_VEL
LIN {X 0,Y 475.127,Z 445.018,A -85,B 0,C 180,E1 -7432.665,E2 -7432.665} C_VEL
LIN {X 0,Y 474.942,Z 453.176,A -85,B 0,C 180,E1 -7435.962,E2 -7435.962} C_VEL
LIN {X 0,Y 474.814,Z 461.049,A -85,B 0,C 180,E1 -7439.148,E2 -7439.148} C_VEL
LIN {X 0,Y 474.683,Z 468.562,A -85,B 0,C 180,E1 -7442.2,E2 -7442.2} C_VEL
LIN {X 0,Y 474.51,Z 476.385,A -85,B 0,C 180,E1 -7445.332,E2 -7445.332} C_VEL
LIN {X 0,Y 473.805,Z 478.174,A -85,B 0,C 180,E1 -7446.007,E2 -7446.007} C_VEL
LIN {X 0,Y 470.913,Z 481.281,A -85,B 0,C 180,E1 -7447.093,E2 -7447.093} C_VEL
LIN {X 0,Y 468.477,Z 483.797,A -85,B 0,C 180,E1 -7447.968,E2 -7447.968} C_VEL
LIN {X 0,Y 467.42,Z 485.66,A -85,B 0,C 180,E1 -7448.647,E2 -7448.647} C_VEL
LIN {X 0,Y 467.328,Z 486.266,A -85,B 0,C 180,E1 -7448.878,E2 -7448.878} C_VEL
LIN {X 0,Y 467.208,Z 492.969,A -85,B 0,C 180,E1 -7451.42,E2 -7451.42} C_VEL
LIN {X 0,Y 470.578,Z 507.99,A -85,B 0,C 180,E1 -7451.897,E2 -7451.897} C_VEL
LIN {X 0,Y 471.844,Z 515.558,A -85,B 0,C 180,E1 -7452.193,E2 -7452.193} C_VEL
LIN {X 0,Y 471.308,Z 529.597,A -85,B 0,C 180,E1 -7452.778,E2 -7452.778} C_VEL
LIN {X 0,Y 470.738,Z 542.899,A -85,B 0,C 180,E1 -7453.52,E2 -7453.52} C_VEL
LIN {X 0,Y 470.089,Z 555.191,A -85,B 0,C 180,E1 -7454.388,E2 -7454.388} C_VEL
LIN {X 0,Y 469.456,Z 566.452,A -85,B 0,C 180,E1 -7455.366,E2 -7455.366} C_VEL
LIN {X 0,Y 468.732,Z 577.768,A -85,B 0,C 180,E1 -7456.561,E2 -7456.561} C_VEL
LIN {X 0,Y 468.224,Z 587.907,A -85,B 0,C 180,E1 -7457.869,E2 -7457.869} C_VEL
LIN {X 0,Y 467.675,Z 596.282,A -85,B 0,C 180,E1 -7459.172,E2 -7459.172} C_VEL
LIN {X 0,Y 467.27,Z 604.279,A -85,B 0,C 180,E1 -7460.694,E2 -7460.694} C_VEL
LIN {X 0,Y 466.985,Z 610.717,A -85,B 0,C 180,E1 -7462.214,E2 -7462.214} C_VEL
LIN {X 0,Y 466.804,Z 616.417,A -85,B 0,C 180,E1 -7463.949,E2 -7463.949} C_VEL
LIN {X 0,Y 466.772,Z 618.675,A -85,B 0,C 180,E1 -7464.816,E2 -7464.816} C_VEL
LIN {X 0,Y 466.684,Z 622.095,A -85,B 0,C 180,E1 -7466.545,E2 -7466.545} C_VEL
LIN {X 0,Y 466.603,Z 624.134,A -85,B 0,C 180,E1 -7468.273,E2 -7468.273} C_VEL
LIN {X 0,Y 466.598,Z 624.84,A -85,B 0,C 180,E1 -7469.999,E2 -7469.999} C_VEL
LIN {X 0,Y 466.601,Z 624.218,A -85,B 0,C 180,E1 -7471.725,E2 -7471.725} C_VEL
LIN {X 0,Y 466.683,Z 622.252,A -85,B 0,C 180,E1 -7473.452,E2 -7473.452} C_VEL
LIN {X 0,Y 466.771,Z 618.901,A -85,B 0,C 180,E1 -7475.182,E2 -7475.182} C_VEL
LIN {X 0,Y 466.849,Z 614.067,A -85,B 0,C 180,E1 -7476.916,E2 -7476.916} C_VEL
LIN {X 0,Y 467.106,Z 607.609,A -85,B 0,C 180,E1 -7478.652,E2 -7478.652} C_VEL
LIN {X 0,Y 467.461,Z 600.411,A -85,B 0,C 180,E1 -7480.174,E2 -7480.174} C_VEL
LIN {X 0,Y 468.012,Z 591.449,A -85,B 0,C 180,E1 -7481.695,E2 -7481.695} C_VEL
LIN {X 0,Y 468.443,Z 582.075,A -85,B 0,C 180,E1 -7483.004,E2 -7483.004} C_VEL
LIN {X 0,Y 469.139,Z 571.698,A -85,B 0,C 180,E1 -7484.199,E2 -7484.199} C_VEL
LIN {X 0,Y 469.763,Z 560.258,A -85,B 0,C 180,E1 -7485.287,E2 -7485.287} C_VEL
LIN {X 0,Y 470.522,Z 547.589,A -85,B 0,C 180,E1 -7486.263,E2 -7486.263} C_VEL
LIN {X 0,Y 471.133,Z 534.651,A -85,B 0,C 180,E1 -7487.055,E2 -7487.055} C_VEL
LIN {X 0,Y 471.616,Z 520.44,A -85,B 0,C 180,E1 -7487.716,E2 -7487.716} C_VEL
LIN {X 0,Y 471.756,Z 514.473,A -85,B 0,C 180,E1 -7487.938,E2 -7487.938} C_VEL
LIN {X 0,Y 469,Z 500.858,A -85,B 0,C 180,E1 -7488.441,E2 -7488.441} C_VEL
LIN {X 0,Y 467.202,Z 492.961,A -85,B 0,C 180,E1 -7488.679,E2 -7488.679} C_VEL
LIN {X 0,Y 467.346,Z 485.222,A -85,B 0,C 180,E1 -7491.617,E2 -7491.617} C_VEL
LIN {X 0,Y 467.485,Z 476.895,A -85,B 0,C 180,E1 -7494.893,E2 -7494.893} C_VEL
LIN {X 0,Y 467.666,Z 468.609,A -85,B 0,C 180,E1 -7498.252,E2 -7498.252} C_VEL
LIN {X 0,Y 467.784,Z 461.722,A -85,B 0,C 180,E1 -7501.088,E2 -7501.088} C_VEL
LIN {X 0,Y 467.979,Z 453.835,A -85,B 0,C 180,E1 -7504.312,E2 -7504.312} C_VEL
LIN {X 0,Y 468.14,Z 446.543,A -85,B 0,C 180,E1 -7507.281,E2 -7507.281} C_VEL
LIN {X 0,Y 467.802,Z 441.319,A -85,B 0,C 180,E1 -7509.399,E2 -7509.399} C_VEL
LIN {X 0,Y 467.66,Z 440.859,A -85,B 0,C 180,E1 -7509.692,E2 -7509.692} C_VEL
LIN {X 0,Y 467.613,Z 440.866,A -85,B 0,C 180,E1 -7512.57,E2 -7512.57} C_VEL
LIN {X 0,Y 467.568,Z 440.871,A -85,B 0,C 180,E1 -7516.175,E2 -7516.175} C_VEL
LIN {X 0,Y 467.583,Z 440.866,A -85,B 0,C 180,E1 -7518.72,E2 -7518.72} C_VEL
LIN {X 0,Y 467.567,Z 440.871,A -85,B 0,C 180,E1 -7521.406,E2 -7521.406} C_VEL
LIN {X 0,Y 467.555,Z 440.869,A -85,B 0,C 180,E1 -7524.259,E2 -7524.259} C_VEL
LIN {X 0,Y 467.574,Z 440.866,A -85,B 0,C 180,E1 -7527.32,E2 -7527.32} C_VEL
LIN {X 0,Y 467.569,Z 440.867,A -85,B 0,C 180,E1 -7530.665,E2 -7530.665} C_VEL
LIN {X 0,Y 467.618,Z 440.859,A -85,B 0,C 180,E1 -7533.2,E2 -7533.2} C_VEL
LIN {X 0,Y 467.584,Z 440.865,A -85,B 0,C 180,E1 -7536.467,E2 -7536.467} C_VEL
LIN {X 0,Y 467.616,Z 440.859,A -85,B 0,C 180,E1 -7539.777,E2 -7539.777} C_VEL
LIN {X 0,Y 467.599,Z 440.863,A -85,B 0,C 180,E1 -7542.506,E2 -7542.506} C_VEL
LIN {X 0,Y 467.596,Z 440.863,A -85,B 0,C 180,E1 -7545.196,E2 -7545.196} C_VEL
LIN {X 0,Y 467.673,Z 440.851,A -85,B 0,C 180,E1 -7547.855,E2 -7547.855} C_VEL
LIN {X 0,Y 467.673,Z 440.851,A -85,B 0,C 180,E1 -7551.357,E2 -7551.357} C_VEL
LIN {X 0,Y 467.744,Z 440.847,A -85,B 0,C 180,E1 -7553.963,E2 -7553.963} C_VEL
LIN {X 0,Y 467.851,Z 440.833,A -85,B 0,C 180,E1 -7557.417,E2 -7557.417} C_VEL
LIN {X 0,Y 467.872,Z 440.829,A -85,B 0,C 180,E1 -7560,E2 -7560} C_VEL
LIN {X 0,Y 467.851,Z 440.829,A -85,B 0,C 180,E1 -7562.583,E2 -7562.583} C_VEL
LIN {X 0,Y 467.734,Z 440.845,A -85,B 0,C 180,E1 -7566.037,E2 -7566.037} C_VEL
LIN {X 0,Y 467.672,Z 440.85,A -85,B 0,C 180,E1 -7568.643,E2 -7568.643} C_VEL
LIN {X 0,Y 467.68,Z 440.849,A -85,B 0,C 180,E1 -7572.379,E2 -7572.379} C_VEL
LIN {X 0,Y 467.638,Z 440.854,A -85,B 0,C 180,E1 -7575.886,E2 -7575.886} C_VEL
LIN {X 0,Y 467.613,Z 440.858,A -85,B 0,C 180,E1 -7579.308,E2 -7579.308} C_VEL
LIN {X 0,Y 467.528,Z 440.873,A -85,B 0,C 180,E1 -7582.074,E2 -7582.074} C_VEL
LIN {X 0,Y 467.593,Z 440.863,A -85,B 0,C 180,E1 -7584.888,E2 -7584.888} C_VEL
LIN {X 0,Y 467.618,Z 440.859,A -85,B 0,C 180,E1 -7587.769,E2 -7587.769} C_VEL
LIN {X 0,Y 467.563,Z 440.867,A -85,B 0,C 180,E1 -7591.047,E2 -7591.047} C_VEL
LIN {X 0,Y 467.581,Z 440.869,A -85,B 0,C 180,E1 -7594.244,E2 -7594.244} C_VEL
LIN {X 0,Y 467.543,Z 440.87,A -85,B 0,C 180,E1 -7597.188,E2 -7597.188} C_VEL
LIN {X 0,Y 467.59,Z 440.864,A -85,B 0,C 180,E1 -7600.263,E2 -7600.263} C_VEL
LIN {X 0,Y 467.611,Z 440.864,A -85,B 0,C 180,E1 -7602.572,E2 -7602.572} C_VEL
LIN {X 0,Y 467.563,Z 440.868,A -85,B 0,C 180,E1 -7605.054,E2 -7605.054} C_VEL
LIN {X 0,Y 467.581,Z 440.867,A -85,B 0,C 180,E1 -7607.441,E2 -7607.441} C_VEL
LIN {X 0,Y 467.613,Z 440.863,A -85,B 0,C 180,E1 -7610.86,E2 -7610.86} C_VEL
LIN {X 0,Y 467.581,Z 440.965,A -85,B 0,C 180,E1 -7612.475,E2 -7612.475} C_VEL
LIN {X 0,Y 469.451,Z 450.355,A -85,B 0,C 180,E1 -7615.932,E2 -7615.932} C_VEL
LIN {X 0,Y 469.911,Z 454.639,A -85,B 0,C 180,E1 -7617.426,E2 -7617.426} C_VEL
LIN {X 0,Y 469.343,Z 463.37,A -85,B 0,C 180,E1 -7620.285,E2 -7620.285} C_VEL
LIN {X 0,Y 468.813,Z 472.791,A -85,B 0,C 180,E1 -7623.275,E2 -7623.275} C_VEL
LIN {X 0,Y 468.301,Z 482.451,A -85,B 0,C 180,E1 -7626.27,E2 -7626.27} C_VEL
LIN {X 0,Y 467.869,Z 492.586,A -85,B 0,C 180,E1 -7629.33,E2 -7629.33} C_VEL
LIN {X 0,Y 467.589,Z 500.085,A -85,B 0,C 180,E1 -7631.55,E2 -7631.55} C_VEL
LIN {X 0,Y 470.435,Z 515.885,A -85,B 0,C 180,E1 -7632.033,E2 -7632.033} C_VEL
LIN {X 0,Y 471.407,Z 521.854,A -85,B 0,C 180,E1 -7632.262,E2 -7632.262} C_VEL
LIN {X 0,Y 470.906,Z 535.655,A -85,B 0,C 180,E1 -7632.827,E2 -7632.827} C_VEL
LIN {X 0,Y 470.357,Z 548.268,A -85,B 0,C 180,E1 -7633.508,E2 -7633.508} C_VEL
LIN {X 0,Y 469.708,Z 561.033,A -85,B 0,C 180,E1 -7634.377,E2 -7634.377} C_VEL
LIN {X 0,Y 468.992,Z 573.857,A -85,B 0,C 180,E1 -7635.464,E2 -7635.464} C_VEL
LIN {X 0,Y 468.429,Z 584.349,A -85,B 0,C 180,E1 -7636.554,E2 -7636.554} C_VEL
LIN {X 0,Y 467.955,Z 594.721,A -85,B 0,C 180,E1 -7637.864,E2 -7637.864} C_VEL
LIN {X 0,Y 467.437,Z 604.557,A -85,B 0,C 180,E1 -7639.388,E2 -7639.388} C_VEL
LIN {X 0,Y 467.134,Z 611.472,A -85,B 0,C 180,E1 -7640.694,E2 -7640.694} C_VEL
LIN {X 0,Y 466.854,Z 618.145,A -85,B 0,C 180,E1 -7642.214,E2 -7642.214} C_VEL
LIN {X 0,Y 466.81,Z 622.738,A -85,B 0,C 180,E1 -7643.542,E2 -7643.542} C_VEL
LIN {X 0,Y 466.761,Z 626.256,A -85,B 0,C 180,E1 -7644.818,E2 -7644.818} C_VEL
LIN {X 0,Y 466.641,Z 628.218,A -85,B 0,C 180,E1 -7645.682,E2 -7645.682} C_VEL
LIN {X 0,Y 466.713,Z 629.749,A -85,B 0,C 180,E1 -7646.548,E2 -7646.548} C_VEL
LIN {X 0,Y 466.655,Z 631.773,A -85,B 0,C 180,E1 -7648.275,E2 -7648.275} C_VEL
LIN {X 0,Y 466.597,Z 632.464,A -85,B 0,C 180,E1 -7650.001,E2 -7650.001} C_VEL
LIN {X 0,Y 466.668,Z 631.736,A -85,B 0,C 180,E1 -7651.727,E2 -7651.727} C_VEL
LIN {X 0,Y 466.662,Z 630.875,A -85,B 0,C 180,E1 -7652.591,E2 -7652.591} C_VEL
LIN {X 0,Y 466.645,Z 627.993,A -85,B 0,C 180,E1 -7654.32,E2 -7654.32} C_VEL
LIN {X 0,Y 466.766,Z 624.907,A -85,B 0,C 180,E1 -7655.618,E2 -7655.618} C_VEL
LIN {X 0,Y 466.826,Z 619.536,A -85,B 0,C 180,E1 -7657.353,E2 -7657.353} C_VEL
LIN {X 0,Y 467.033,Z 614.379,A -85,B 0,C 180,E1 -7658.656,E2 -7658.656} C_VEL
LIN {X 0,Y 467.288,Z 606.966,A -85,B 0,C 180,E1 -7660.18,E2 -7660.18} C_VEL
LIN {X 0,Y 467.693,Z 599.183,A -85,B 0,C 180,E1 -7661.486,E2 -7661.486} C_VEL
LIN {X 0,Y 468.18,Z 589.267,A -85,B 0,C 180,E1 -7662.856,E2 -7662.856} C_VEL
LIN {X 0,Y 468.81,Z 578.254,A -85,B 0,C 180,E1 -7664.1,E2 -7664.1} C_VEL
LIN {X 0,Y 469.392,Z 566.462,A -85,B 0,C 180,E1 -7665.191,E2 -7665.191} C_VEL
LIN {X 0,Y 470,Z 554.871,A -85,B 0,C 180,E1 -7666.06,E2 -7666.06} C_VEL
LIN {X 0,Y 470.547,Z 543.135,A -85,B 0,C 180,E1 -7666.77,E2 -7666.77} C_VEL
LIN {X 0,Y 471.036,Z 529.31,A -85,B 0,C 180,E1 -7667.419,E2 -7667.419} C_VEL
LIN {X 0,Y 471.178,Z 520.742,A -85,B 0,C 180,E1 -7667.729,E2 -7667.729} C_VEL
LIN {X 0,Y 468.237,Z 503.175,A -85,B 0,C 180,E1 -7668.309,E2 -7668.309} C_VEL
LIN {X 0,Y 467.561,Z 499.437,A -85,B 0,C 180,E1 -7668.432,E2 -7668.432} C_VEL
LIN {X 0,Y 467.947,Z 488.682,A -85,B 0,C 180,E1 -7671.652,E2 -7671.652} C_VEL
LIN {X 0,Y 468.431,Z 478.554,A -85,B 0,C 180,E1 -7674.841,E2 -7674.841} C_VEL
LIN {X 0,Y 469.097,Z 469.53,A -85,B 0,C 180,E1 -7677.879,E2 -7677.879} C_VEL
LIN {X 0,Y 469.99,Z 460.914,A -85,B 0,C 180,E1 -7681.058,E2 -7681.058} C_VEL
LIN {X 0,Y 470.487,Z 457.276,A -85,B 0,C 180,E1 -7682.532,E2 -7682.532} C_VEL
LIN {X 0,Y 470.24,Z 453.931,A -85,B 0,C 180,E1 -7684.088,E2 -7684.088} C_VEL
LIN {X 0,Y 469.261,Z 449.128,A -85,B 0,C 180,E1 -7686.804,E2 -7686.804} C_VEL
LIN {X 0,Y 468.678,Z 446.072,A -85,B 0,C 180,E1 -7689.037,E2 -7689.037} C_VEL
LIN {X 0,Y 468.21,Z 443.832,A -85,B 0,C 180,E1 -7691.365,E2 -7691.365} C_VEL
LIN {X 0,Y 467.882,Z 442.592,A -85,B 0,C 180,E1 -7693.863,E2 -7693.863} C_VEL
LIN {X 0,Y 467.889,Z 442.446,A -85,B 0,C 180,E1 -7696.295,E2 -7696.295} C_VEL
LIN {X 0,Y 468.063,Z 443.264,A -85,B 0,C 180,E1 -7698.657,E2 -7698.657} C_VEL
LIN {X 0,Y 468.398,Z 445.135,A -85,B 0,C 180,E1 -7701.282,E2 -7701.282} C_VEL
LIN {X 0,Y 468.711,Z 447.996,A -85,B 0,C 180,E1 -7704.067,E2 -7704.067} C_VEL
LIN {X 0,Y 468.49,Z 450.868,A -85,B 0,C 180,E1 -7706.286,E2 -7706.286} C_VEL
LIN {X 0,Y 468.116,Z 455.27,A -85,B 0,C 180,E1 -7709.306,E2 -7709.306} C_VEL
LIN {X 0,Y 467.816,Z 460.22,A -85,B 0,C 180,E1 -7712.42,E2 -7712.42} C_VEL
LIN {X 0,Y 467.558,Z 464.73,A -85,B 0,C 180,E1 -7715.11,E2 -7715.11} C_VEL
LIN {X 0,Y 467.389,Z 469.638,A -85,B 0,C 180,E1 -7717.919,E2 -7717.919} C_VEL
LIN {X 0,Y 467.183,Z 475.916,A -85,B 0,C 180,E1 -7721.395,E2 -7721.395} C_VEL
LIN {X 0,Y 467.091,Z 481.572,A -85,B 0,C 180,E1 -7724.437,E2 -7724.437} C_VEL
LIN {X 0,Y 469.959,Z 494.547,A -85,B 0,C 180,E1 -7724.968,E2 -7724.968} C_VEL
LIN {X 0,Y 470.512,Z 499.39,A -85,B 0,C 180,E1 -7725.189,E2 -7725.189} C_VEL
LIN {X 0,Y 470.047,Z 512.243,A -85,B 0,C 180,E1 -7725.828,E2 -7725.828} C_VEL
LIN {X 0,Y 469.521,Z 524.773,A -85,B 0,C 180,E1 -7726.645,E2 -7726.645} C_VEL
LIN {X 0,Y 469.039,Z 535.824,A -85,B 0,C 180,E1 -7727.561,E2 -7727.561} C_VEL
LIN {X 0,Y 468.515,Z 545.411,A -85,B 0,C 180,E1 -7728.536,E2 -7728.536} C_VEL
LIN {X 0,Y 468.028,Z 554.233,A -85,B 0,C 180,E1 -7729.619,E2 -7729.619} C_VEL
LIN {X 0,Y 467.624,Z 562.899,A -85,B 0,C 180,E1 -7730.92,E2 -7730.92} C_VEL
LIN {X 0,Y 467.258,Z 569.83,A -85,B 0,C 180,E1 -7732.22,E2 -7732.22} C_VEL
LIN {X 0,Y 467.092,Z 575.487,A -85,B 0,C 180,E1 -7733.552,E2 -7733.552} C_VEL
LIN {X 0,Y 466.802,Z 579.733,A -85,B 0,C 180,E1 -7734.817,E2 -7734.817} C_VEL
LIN {X 0,Y 466.901,Z 582.021,A -85,B 0,C 180,E1 -7735.684,E2 -7735.684} C_VEL
LIN {X 0,Y 466.786,Z 583.892,A -85,B 0,C 180,E1 -7736.547,E2 -7736.547} C_VEL
LIN {X 0,Y 466.751,Z 585.3,A -85,B 0,C 180,E1 -7737.411,E2 -7737.411} C_VEL
LIN {X 0,Y 466.698,Z 586.289,A -85,B 0,C 180,E1 -7738.274,E2 -7738.274} C_VEL
LIN {X 0,Y 466.599,Z 587.1,A -85,B 0,C 180,E1 -7740,E2 -7740} C_VEL
LIN {X 0,Y 466.621,Z 586.881,A -85,B 0,C 180,E1 -7740.863,E2 -7740.863} C_VEL
LIN {X 0,Y 466.697,Z 586.252,A -85,B 0,C 180,E1 -7741.726,E2 -7741.726} C_VEL
LIN {X 0,Y 466.737,Z 585.236,A -85,B 0,C 180,E1 -7742.589,E2 -7742.589} C_VEL
LIN {X 0,Y 466.785,Z 583.822,A -85,B 0,C 180,E1 -7743.453,E2 -7743.453} C_VEL
LIN {X 0,Y 466.81,Z 580.862,A -85,B 0,C 180,E1 -7744.75,E2 -7744.75} C_VEL
LIN {X 0,Y 467.015,Z 576.859,A -85,B 0,C 180,E1 -7746.047,E2 -7746.047} C_VEL
LIN {X 0,Y 467.138,Z 570.721,A -85,B 0,C 180,E1 -7747.565,E2 -7747.565} C_VEL
LIN {X 0,Y 467.463,Z 564.012,A -85,B 0,C 180,E1 -7748.865,E2 -7748.865} C_VEL
LIN {X 0,Y 467.83,Z 555.708,A -85,B 0,C 180,E1 -7750.167,E2 -7750.167} C_VEL
LIN {X 0,Y 468.215,Z 547.23,A -85,B 0,C 180,E1 -7751.253,E2 -7751.253} C_VEL
LIN {X 0,Y 468.84,Z 536.805,A -85,B 0,C 180,E1 -7752.334,E2 -7752.334} C_VEL
LIN {X 0,Y 469.315,Z 525.171,A -85,B 0,C 180,E1 -7753.311,E2 -7753.311} C_VEL
LIN {X 0,Y 469.767,Z 513.711,A -85,B 0,C 180,E1 -7754.07,E2 -7754.07} C_VEL
LIN {X 0,Y 470.215,Z 500.855,A -85,B 0,C 180,E1 -7754.72,E2 -7754.72} C_VEL
LIN {X 0,Y 470.006,Z 496.059,A -85,B 0,C 180,E1 -7754.926,E2 -7754.926} C_VEL
LIN {X 0,Y 467.544,Z 483.699,A -85,B 0,C 180,E1 -7755.413,E2 -7755.413} C_VEL
LIN {X 0,Y 466.914,Z 480.492,A -85,B 0,C 180,E1 -7755.518,E2 -7755.518} C_VEL
LIN {X 0,Y 467.042,Z 474.6,A -85,B 0,C 180,E1 -7758.554,E2 -7758.554} C_VEL
LIN {X 0,Y 467.158,Z 467.823,A -85,B 0,C 180,E1 -7762.093,E2 -7762.093} C_VEL
LIN {X 0,Y 467.264,Z 462.525,A -85,B 0,C 180,E1 -7764.907,E2 -7764.907} C_VEL
LIN {X 0,Y 467.434,Z 457.197,A -85,B 0,C 180,E1 -7767.781,E2 -7767.781} C_VEL
LIN {X 0,Y 467.582,Z 451.81,A -85,B 0,C 180,E1 -7770.733,E2 -7770.733} C_VEL
LIN {X 0,Y 467.755,Z 446.374,A -85,B 0,C 180,E1 -7773.775,E2 -7773.775} C_VEL
LIN {X 0,Y 467.741,Z 441.784,A -85,B 0,C 180,E1 -7776.406,E2 -7776.406} C_VEL
LIN {X 0,Y 467.6,Z 440.867,A -85,B 0,C 180,E1 -7776.956,E2 -7776.956} C_VEL
LIN {X 0,Y 467.584,Z 440.866,A -85,B 0,C 180,E1 -7780.264,E2 -7780.264} C_VEL
LIN {X 0,Y 467.592,Z 440.866,A -85,B 0,C 180,E1 -7782.567,E2 -7782.567} C_VEL
LIN {X 0,Y 467.576,Z 440.871,A -85,B 0,C 180,E1 -7785.053,E2 -7785.053} C_VEL
LIN {X 0,Y 467.594,Z 440.87,A -85,B 0,C 180,E1 -7787.44,E2 -7787.44} C_VEL
LIN {X 0,Y 467.659,Z 440.905,A -85,B 0,C 180,E1 -7790.514,E2 -7790.514} C_VEL
LIN {X 0,Y 468.1,Z 444.543,A -85,B 0,C 180,E1 -7792.006,E2 -7792.006} C_VEL
LIN {X 0,Y 467.989,Z 451.139,A -85,B 0,C 180,E1 -7794.691,E2 -7794.691} C_VEL
LIN {X 0,Y 467.836,Z 458.68,A -85,B 0,C 180,E1 -7797.777,E2 -7797.777} C_VEL
LIN {X 0,Y 467.72,Z 465.641,A -85,B 0,C 180,E1 -7800.635,E2 -7800.635} C_VEL
LIN {X 0,Y 467.558,Z 473.104,A -85,B 0,C 180,E1 -7803.677,E2 -7803.677} C_VEL
LIN {X 0,Y 467.362,Z 481.403,A -85,B 0,C 180,E1 -7806.984,E2 -7806.984} C_VEL
LIN {X 0,Y 467.328,Z 486.266,A -85,B 0,C 180,E1 -7808.878,E2 -7808.878} C_VEL
LIN {X 0,Y 466.376,Z 487.114,A -85,B 0,C 180,E1 -7809.163,E2 -7809.163} C_VEL
LIN {X 0,Y 460.749,Z 489.444,A -85,B 0,C 180,E1 -7809.814,E2 -7809.814} C_VEL
LIN {X 0,Y 460.21,Z 490.067,A -85,B 0,C 180,E1 -7810.029,E2 -7810.029} C_VEL
LIN {X 0,Y 460.175,Z 492.965,A -85,B 0,C 180,E1 -7811.127,E2 -7811.127} C_VEL
LIN {X 0,Y 463.514,Z 507.972,A -85,B 0,C 180,E1 -7811.61,E2 -7811.61} C_VEL
LIN {X 0,Y 465.077,Z 516.31,A -85,B 0,C 180,E1 -7811.953,E2 -7811.953} C_VEL
LIN {X 0,Y 464.564,Z 528.74,A -85,B 0,C 180,E1 -7812.473,E2 -7812.473} C_VEL
LIN {X 0,Y 464.036,Z 541.485,A -85,B 0,C 180,E1 -7813.178,E2 -7813.178} C_VEL
LIN {X 0,Y 463.318,Z 553.853,A -85,B 0,C 180,E1 -7814.041,E2 -7814.041} C_VEL
LIN {X 0,Y 462.63,Z 565.357,A -85,B 0,C 180,E1 -7815.033,E2 -7815.033} C_VEL
LIN {X 0,Y 461.921,Z 575.912,A -85,B 0,C 180,E1 -7816.134,E2 -7816.134} C_VEL
LIN {X 0,Y 461.293,Z 585.515,A -85,B 0,C 180,E1 -7817.34,E2 -7817.34} C_VEL
LIN {X 0,Y 460.903,Z 593.681,A -85,B 0,C 180,E1 -7818.566,E2 -7818.566} C_VEL
LIN {X 0,Y 460.395,Z 602.197,A -85,B 0,C 180,E1 -7820.11,E2 -7820.11} C_VEL
LIN {X 0,Y 460.03,Z 609.068,A -85,B 0,C 180,E1 -7821.654,E2 -7821.654} C_VEL
LIN {X 0,Y 459.795,Z 613.827,A -85,B 0,C 180,E1 -7822.975,E2 -7822.975} C_VEL
LIN {X 0,Y 459.708,Z 618.73,A -85,B 0,C 180,E1 -7824.736,E2 -7824.736} C_VEL
LIN {X 0,Y 459.581,Z 622.151,A -85,B 0,C 180,E1 -7826.492,E2 -7826.492} C_VEL
LIN {X 0,Y 459.516,Z 624.19,A -85,B 0,C 180,E1 -7828.246,E2 -7828.246} C_VEL
LIN {X 0,Y 459.5,Z 624.896,A -85,B 0,C 180,E1 -7829.999,E2 -7829.999} C_VEL
LIN {X 0,Y 459.514,Z 624.273,A -85,B 0,C 180,E1 -7831.752,E2 -7831.752} C_VEL
LIN {X 0,Y 459.58,Z 622.305,A -85,B 0,C 180,E1 -7833.506,E2 -7833.506} C_VEL
LIN {X 0,Y 459.707,Z 618.953,A -85,B 0,C 180,E1 -7835.262,E2 -7835.262} C_VEL
LIN {X 0,Y 459.77,Z 614.119,A -85,B 0,C 180,E1 -7837.023,E2 -7837.023} C_VEL
LIN {X 0,Y 460.064,Z 607.659,A -85,B 0,C 180,E1 -7838.786,E2 -7838.786} C_VEL
LIN {X 0,Y 460.435,Z 600.459,A -85,B 0,C 180,E1 -7840.331,E2 -7840.331} C_VEL
LIN {X 0,Y 461.031,Z 591.496,A -85,B 0,C 180,E1 -7841.875,E2 -7841.875} C_VEL
LIN {X 0,Y 461.501,Z 582.12,A -85,B 0,C 180,E1 -7843.203,E2 -7843.203} C_VEL
LIN {X 0,Y 462.221,Z 571.74,A -85,B 0,C 180,E1 -7844.416,E2 -7844.416} C_VEL
LIN {X 0,Y 462.888,Z 560.296,A -85,B 0,C 180,E1 -7845.52,E2 -7845.52} C_VEL
LIN {X 0,Y 463.689,Z 547.621,A -85,B 0,C 180,E1 -7846.509,E2 -7846.509} C_VEL
LIN {X 0,Y 464.37,Z 534.08,A -85,B 0,C 180,E1 -7847.344,E2 -7847.344} C_VEL
LIN {X 0,Y 464.892,Z 520.094,A -85,B 0,C 180,E1 -7847.995,E2 -7847.995} C_VEL
LIN {X 0,Y 464.905,Z 515.202,A -85,B 0,C 180,E1 -7848.187,E2 -7848.187} C_VEL
LIN {X 0,Y 462.088,Z 501.221,A -85,B 0,C 180,E1 -7848.718,E2 -7848.718} C_VEL
LIN {X 0,Y 460.16,Z 492.9,A -85,B 0,C 180,E1 -7848.992,E2 -7848.992} C_VEL
LIN {X 0,Y 460.301,Z 485.136,A -85,B 0,C 180,E1 -7851.966,E2 -7851.966} C_VEL
LIN {X 0,Y 460.439,Z 476.754,A -85,B 0,C 180,E1 -7855.3,E2 -7855.3} C_VEL
LIN {X 0,Y 460.623,Z 469.595,A -85,B 0,C 180,E1 -7858.227,E2 -7858.227} C_VEL
LIN {X 0,Y 460.753,Z 462.365,A -85,B 0,C 180,E1 -7861.238,E2 -7861.238} C_VEL
LIN {X 0,Y 460.94,Z 454.265,A -85,B 0,C 180,E1 -7864.579,E2 -7864.579} C_VEL
LIN {X 0,Y 461.119,Z 446.987,A -85,B 0,C 180,E1 -7867.576,E2 -7867.576} C_VEL
LIN {X 0,Y 460.829,Z 442.656,A -85,B 0,C 180,E1 -7869.357,E2 -7869.357} C_VEL
LIN {X 0,Y 460.613,Z 441.737,A -85,B 0,C 180,E1 -7869.852,E2 -7869.852} C_VEL
LIN {X 0,Y 460.518,Z 441.746,A -85,B 0,C 180,E1 -7873.371,E2 -7873.371} C_VEL
LIN {X 0,Y 460.518,Z 441.748,A -85,B 0,C 180,E1 -7876.627,E2 -7876.627} C_VEL
LIN {X 0,Y 460.551,Z 441.743,A -85,B 0,C 180,E1 -7879.727,E2 -7879.727} C_VEL
LIN {X 0,Y 460.52,Z 441.744,A -85,B 0,C 180,E1 -7882.518,E2 -7882.518} C_VEL
LIN {X 0,Y 460.54,Z 441.739,A -85,B 0,C 180,E1 -7885.623,E2 -7885.623} C_VEL
LIN {X 0,Y 460.528,Z 441.74,A -85,B 0,C 180,E1 -7888.744,E2 -7888.744} C_VEL
LIN {X 0,Y 460.549,Z 441.744,A -85,B 0,C 180,E1 -7891.767,E2 -7891.767} C_VEL
LIN {X 0,Y 460.551,Z 441.739,A -85,B 0,C 180,E1 -7894.705,E2 -7894.705} C_VEL
LIN {X 0,Y 460.519,Z 441.738,A -85,B 0,C 180,E1 -7897.572,E2 -7897.572} C_VEL
LIN {X 0,Y 460.56,Z 441.744,A -85,B 0,C 180,E1 -7900.384,E2 -7900.384} C_VEL
LIN {X 0,Y 460.62,Z 441.734,A -85,B 0,C 180,E1 -7904.059,E2 -7904.059} C_VEL
LIN {X 0,Y 460.619,Z 441.731,A -85,B 0,C 180,E1 -7907.666,E2 -7907.666} C_VEL
LIN {X 0,Y 460.62,Z 441.73,A -85,B 0,C 180,E1 -7911.224,E2 -7911.224} C_VEL
LIN {X 0,Y 460.708,Z 441.722,A -85,B 0,C 180,E1 -7913.87,E2 -7913.87} C_VEL
LIN {X 0,Y 460.816,Z 441.709,A -85,B 0,C 180,E1 -7917.378,E2 -7917.378} C_VEL
LIN {X 0,Y 460.843,Z 441.704,A -85,B 0,C 180,E1 -7920,E2 -7920} C_VEL
LIN {X 0,Y 460.816,Z 441.704,A -85,B 0,C 180,E1 -7922.622,E2 -7922.622} C_VEL
LIN {X 0,Y 460.7,Z 441.722,A -85,B 0,C 180,E1 -7926.13,E2 -7926.13} C_VEL
LIN {X 0,Y 460.619,Z 441.728,A -85,B 0,C 180,E1 -7928.776,E2 -7928.776} C_VEL
LIN {X 0,Y 460.623,Z 441.728,A -85,B 0,C 180,E1 -7932.457,E2 -7932.457} C_VEL
LIN {X 0,Y 460.589,Z 441.732,A -85,B 0,C 180,E1 -7935.998,E2 -7935.998} C_VEL
LIN {X 0,Y 460.56,Z 441.739,A -85,B 0,C 180,E1 -7938.903,E2 -7938.903} C_VEL
LIN {X 0,Y 460.506,Z 441.747,A -85,B 0,C 180,E1 -7941.486,E2 -7941.486} C_VEL
LIN {X 0,Y 460.533,Z 441.742,A -85,B 0,C 180,E1 -7944.333,E2 -7944.333} C_VEL
LIN {X 0,Y 460.574,Z 441.741,A -85,B 0,C 180,E1 -7947.244,E2 -7947.244} C_VEL
LIN {X 0,Y 460.518,Z 441.747,A -85,B 0,C 180,E1 -7950.239,E2 -7950.239} C_VEL
LIN {X 0,Y 460.52,Z 441.744,A -85,B 0,C 180,E1 -7953.326,E2 -7953.326} C_VEL
LIN {X 0,Y 460.471,Z 441.749,A -85,B 0,C 180,E1 -7956.53,E2 -7956.53} C_VEL
LIN {X 0,Y 460.571,Z 441.739,A -85,B 0,C 180,E1 -7959.858,E2 -7959.858} C_VEL
LIN {X 0,Y 460.535,Z 441.747,A -85,B 0,C 180,E1 -7962.905,E2 -7962.905} C_VEL
LIN {X 0,Y 460.504,Z 441.748,A -85,B 0,C 180,E1 -7965.831,E2 -7965.831} C_VEL
LIN {X 0,Y 460.533,Z 441.745,A -85,B 0,C 180,E1 -7968.991,E2 -7968.991} C_VEL
LIN {X 0,Y 460.531,Z 441.744,A -85,B 0,C 180,E1 -7972.105,E2 -7972.105} C_VEL
LIN {X 0,Y 462.106,Z 449.934,A -85,B 0,C 180,E1 -7975.212,E2 -7975.212} C_VEL
LIN {X 0,Y 462.937,Z 454.519,A -85,B 0,C 180,E1 -7976.873,E2 -7976.873} C_VEL
LIN {X 0,Y 462.663,Z 460.55,A -85,B 0,C 180,E1 -7978.906,E2 -7978.906} C_VEL
LIN {X 0,Y 462.022,Z 469.763,A -85,B 0,C 180,E1 -7981.916,E2 -7981.916} C_VEL
LIN {X 0,Y 461.542,Z 478.708,A -85,B 0,C 180,E1 -7984.765,E2 -7984.765} C_VEL
LIN {X 0,Y 460.983,Z 489.36,A -85,B 0,C 180,E1 -7988.069,E2 -7988.069} C_VEL
LIN {X 0,Y 460.556,Z 499.961,A -85,B 0,C 180,E1 -7991.285,E2 -7991.285} C_VEL
LIN {X 0,Y 463.349,Z 515.157,A -85,B 0,C 180,E1 -7991.76,E2 -7991.76} C_VEL
LIN {X 0,Y 464.497,Z 523.152,A -85,B 0,C 180,E1 -7992.074,E2 -7992.074} C_VEL
LIN {X 0,Y 463.946,Z 537.853,A -85,B 0,C 180,E1 -7992.704,E2 -7992.704} C_VEL
LIN {X 0,Y 463.453,Z 549.806,A -85,B 0,C 180,E1 -7993.369,E2 -7993.369} C_VEL
LIN {X 0,Y 462.747,Z 562.379,A -85,B 0,C 180,E1 -7994.249,E2 -7994.249} C_VEL
LIN {X 0,Y 462.073,Z 573.812,A -85,B 0,C 180,E1 -7995.242,E2 -7995.242} C_VEL
LIN {X 0,Y 461.494,Z 584.287,A -85,B 0,C 180,E1 -7996.348,E2 -7996.348} C_VEL
LIN {X 0,Y 460.942,Z 594.675,A -85,B 0,C 180,E1 -7997.676,E2 -7997.676} C_VEL
LIN {X 0,Y 460.494,Z 603.219,A -85,B 0,C 180,E1 -7999.003,E2 -7999.003} C_VEL
LIN {X 0,Y 460.085,Z 611.354,A -85,B 0,C 180,E1 -8000.55,E2 -8000.55} C_VEL
LIN {X 0,Y 459.797,Z 617.883,A -85,B 0,C 180,E1 -8002.094,E2 -8002.094} C_VEL
LIN {X 0,Y 459.673,Z 623.658,A -85,B 0,C 180,E1 -8003.857,E2 -8003.857} C_VEL
LIN {X 0,Y 459.671,Z 625.952,A -85,B 0,C 180,E1 -8004.738,E2 -8004.738} C_VEL
LIN {X 0,Y 459.609,Z 629.398,A -85,B 0,C 180,E1 -8006.494,E2 -8006.494} C_VEL
LIN {X 0,Y 459.564,Z 631.427,A -85,B 0,C 180,E1 -8008.248,E2 -8008.248} C_VEL
LIN {X 0,Y 459.55,Z 631.971,A -85,B 0,C 180,E1 -8009.125,E2 -8009.125} C_VEL
LIN {X 0,Y 459.551,Z 631.938,A -85,B 0,C 180,E1 -8010.877,E2 -8010.877} C_VEL
LIN {X 0,Y 459.585,Z 630.578,A -85,B 0,C 180,E1 -8012.631,E2 -8012.631} C_VEL
LIN {X 0,Y 459.563,Z 627.841,A -85,B 0,C 180,E1 -8014.386,E2 -8014.386} C_VEL
LIN {X 0,Y 459.684,Z 624.871,A -85,B 0,C 180,E1 -8015.704,E2 -8015.704} C_VEL
LIN {X 0,Y 459.765,Z 619.49,A -85,B 0,C 180,E1 -8017.467,E2 -8017.467} C_VEL
LIN {X 0,Y 459.964,Z 614.341,A -85,B 0,C 180,E1 -8018.79,E2 -8018.79} C_VEL
LIN {X 0,Y 460.258,Z 606.912,A -85,B 0,C 180,E1 -8020.337,E2 -8020.337} C_VEL
LIN {X 0,Y 460.702,Z 599.132,A -85,B 0,C 180,E1 -8021.662,E2 -8021.662} C_VEL
LIN {X 0,Y 461.191,Z 589.404,A -85,B 0,C 180,E1 -8023.03,E2 -8023.03} C_VEL
LIN {X 0,Y 461.9,Z 578.205,A -85,B 0,C 180,E1 -8024.316,E2 -8024.316} C_VEL
LIN {X 0,Y 462.518,Z 566.416,A -85,B 0,C 180,E1 -8025.422,E2 -8025.422} C_VEL
LIN {X 0,Y 463.173,Z 554.83,A -85,B 0,C 180,E1 -8026.304,E2 -8026.304} C_VEL
LIN {X 0,Y 463.816,Z 541.737,A -85,B 0,C 180,E1 -8027.099,E2 -8027.099} C_VEL
LIN {X 0,Y 464.307,Z 527.941,A -85,B 0,C 180,E1 -8027.736,E2 -8027.736} C_VEL
LIN {X 0,Y 464.361,Z 521.553,A -85,B 0,C 180,E1 -8027.972,E2 -8027.972} C_VEL
LIN {X 0,Y 461.607,Z 504.859,A -85,B 0,C 180,E1 -8028.538,E2 -8028.538} C_VEL
LIN {X 0,Y 460.543,Z 499.229,A -85,B 0,C 180,E1 -8028.735,E2 -8028.735} C_VEL
LIN {X 0,Y 460.943,Z 488.803,A -85,B 0,C 180,E1 -8031.935,E2 -8031.935} C_VEL
LIN {X 0,Y 461.503,Z 478.597,A -85,B 0,C 180,E1 -8035.24,E2 -8035.24} C_VEL
LIN {X 0,Y 462.198,Z 470.297,A -85,B 0,C 180,E1 -8038.124,E2 -8038.124} C_VEL
LIN {X 0,Y 463.06,Z 462.548,A -85,B 0,C 180,E1 -8041.067,E2 -8041.067} C_VEL
LIN {X 0,Y 463.589,Z 458.952,A -85,B 0,C 180,E1 -8042.561,E2 -8042.561} C_VEL
LIN {X 0,Y 463.353,Z 455.658,A -85,B 0,C 180,E1 -8044.14,E2 -8044.14} C_VEL
LIN {X 0,Y 462.571,Z 451.756,A -85,B 0,C 180,E1 -8046.366,E2 -8046.366} C_VEL
LIN {X 0,Y 461.871,Z 448.012,A -85,B 0,C 180,E1 -8049.101,E2 -8049.101} C_VEL
LIN {X 0,Y 461.353,Z 445.657,A -85,B 0,C 180,E1 -8051.717,E2 -8051.717} C_VEL
LIN {X 0,Y 461.064,Z 444.55,A -85,B 0,C 180,E1 -8054.24,E2 -8054.24} C_VEL
LIN {X 0,Y 461.066,Z 444.503,A -85,B 0,C 180,E1 -8056.691,E2 -8056.691} C_VEL
LIN {X 0,Y 461.24,Z 445.389,A -85,B 0,C 180,E1 -8059.065,E2 -8059.065} C_VEL
LIN {X 0,Y 461.544,Z 446.969,A -85,B 0,C 180,E1 -8061.368,E2 -8061.368} C_VEL
LIN {X 0,Y 461.77,Z 449.296,A -85,B 0,C 180,E1 -8063.77,E2 -8063.77} C_VEL
LIN {X 0,Y 461.628,Z 451.637,A -85,B 0,C 180,E1 -8065.716,E2 -8065.716} C_VEL
LIN {X 0,Y 461.207,Z 455.884,A -85,B 0,C 180,E1 -8068.795,E2 -8068.795} C_VEL
LIN {X 0,Y 460.846,Z 461.093,A -85,B 0,C 180,E1 -8072.193,E2 -8072.193} C_VEL
LIN {X 0,Y 460.588,Z 465.194,A -85,B 0,C 180,E1 -8074.707,E2 -8074.707} C_VEL
LIN {X 0,Y 460.388,Z 470.051,A -85,B 0,C 180,E1 -8077.565,E2 -8077.565} C_VEL
LIN {X 0,Y 460.197,Z 474.991,A -85,B 0,C 180,E1 -8080.368,E2 -8080.368} C_VEL
LIN {X 0,Y 460.021,Z 481.818,A -85,B 0,C 180,E1 -8084.123,E2 -8084.123} C_VEL
LIN {X 0,Y 463.029,Z 494.966,A -85,B 0,C 180,E1 -8084.701,E2 -8084.701} C_VEL
LIN {X 0,Y 463.693,Z 498.866,A -85,B 0,C 180,E1 -8084.896,E2 -8084.896} C_VEL
LIN {X 0,Y 463.326,Z 511.155,A -85,B 0,C 180,E1 -8085.506,E2 -8085.506} C_VEL
LIN {X 0,Y 462.809,Z 522.731,A -85,B 0,C 180,E1 -8086.248,E2 -8086.248} C_VEL
LIN {X 0,Y 462.254,Z 533.98,A -85,B 0,C 180,E1 -8087.153,E2 -8087.153} C_VEL
LIN {X 0,Y 461.646,Z 543.993,A -85,B 0,C 180,E1 -8088.14,E2 -8088.14} C_VEL
LIN {X 0,Y 461.166,Z 553.088,A -85,B 0,C 180,E1 -8089.241,E2 -8089.241} C_VEL
LIN {X 0,Y 460.685,Z 561.971,A -85,B 0,C 180,E1 -8090.561,E2 -8090.561} C_VEL
LIN {X 0,Y 460.306,Z 569.157,A -85,B 0,C 180,E1 -8091.881,E2 -8091.881} C_VEL
LIN {X 0,Y 460.001,Z 575.169,A -85,B 0,C 180,E1 -8093.263,E2 -8093.263} C_VEL
LIN {X 0,Y 459.883,Z 578.77,A -85,B 0,C 180,E1 -8094.299,E2 -8094.299} C_VEL
LIN {X 0,Y 459.824,Z 582.391,A -85,B 0,C 180,E1 -8095.617,E2 -8095.617} C_VEL
LIN {X 0,Y 459.726,Z 584.26,A -85,B 0,C 180,E1 -8096.494,E2 -8096.494} C_VEL
LIN {X 0,Y 459.669,Z 585.666,A -85,B 0,C 180,E1 -8097.371,E2 -8097.371} C_VEL
LIN {X 0,Y 459.636,Z 586.65,A -85,B 0,C 180,E1 -8098.248,E2 -8098.248} C_VEL
LIN {X 0,Y 459.531,Z 587.451,A -85,B 0,C 180,E1 -8100,E2 -8100} C_VEL
LIN {X 0,Y 459.555,Z 587.222,A -85,B 0,C 180,E1 -8100.876,E2 -8100.876} C_VEL
LIN {X 0,Y 459.635,Z 586.585,A -85,B 0,C 180,E1 -8101.752,E2 -8101.752} C_VEL
LIN {X 0,Y 459.724,Z 584.131,A -85,B 0,C 180,E1 -8103.506,E2 -8103.506} C_VEL
LIN {X 0,Y 459.723,Z 581.151,A -85,B 0,C 180,E1 -8104.823,E2 -8104.823} C_VEL
LIN {X 0,Y 459.96,Z 577.124,A -85,B 0,C 180,E1 -8106.14,E2 -8106.14} C_VEL
LIN {X 0,Y 460.101,Z 570.954,A -85,B 0,C 180,E1 -8107.681,E2 -8107.681} C_VEL
LIN {X 0,Y 460.437,Z 564.219,A -85,B 0,C 180,E1 -8109.001,E2 -8109.001} C_VEL
LIN {X 0,Y 460.841,Z 555.883,A -85,B 0,C 180,E1 -8110.323,E2 -8110.323} C_VEL
LIN {X 0,Y 461.245,Z 547.375,A -85,B 0,C 180,E1 -8111.425,E2 -8111.425} C_VEL
LIN {X 0,Y 461.894,Z 536.96,A -85,B 0,C 180,E1 -8112.519,E2 -8112.519} C_VEL
LIN {X 0,Y 462.377,Z 525.943,A -85,B 0,C 180,E1 -8113.461,E2 -8113.461} C_VEL
LIN {X 0,Y 462.89,Z 513.789,A -85,B 0,C 180,E1 -8114.284,E2 -8114.284} C_VEL
LIN {X 0,Y 463.352,Z 500.944,A -85,B 0,C 180,E1 -8114.943,E2 -8114.943} C_VEL
LIN {X 0,Y 462.951,Z 495.9,A -85,B 0,C 180,E1 -8115.169,E2 -8115.169} C_VEL
LIN {X 0,Y 460.178,Z 482.452,A -85,B 0,C 180,E1 -8115.707,E2 -8115.707} C_VEL
LIN {X 0,Y 459.86,Z 480.63,A -85,B 0,C 180,E1 -8115.773,E2 -8115.773} C_VEL
LIN {X 0,Y 459.97,Z 474.972,A -85,B 0,C 180,E1 -8118.715,E2 -8118.715} C_VEL
LIN {X 0,Y 460.076,Z 469.671,A -85,B 0,C 180,E1 -8121.507,E2 -8121.507} C_VEL
LIN {X 0,Y 460.183,Z 464.362,A -85,B 0,C 180,E1 -8124.353,E2 -8124.353} C_VEL
LIN {X 0,Y 460.356,Z 459.003,A -85,B 0,C 180,E1 -8127.258,E2 -8127.258} C_VEL
LIN {X 0,Y 460.507,Z 453.609,A -85,B 0,C 180,E1 -8130.24,E2 -8130.24} C_VEL
LIN {X 0,Y 460.676,Z 448.168,A -85,B 0,C 180,E1 -8133.313,E2 -8133.313} C_VEL
LIN {X 0,Y 460.747,Z 443.407,A -85,B 0,C 180,E1 -8136.056,E2 -8136.056} C_VEL
LIN {X 0,Y 460.568,Z 441.743,A -85,B 0,C 180,E1 -8137.067,E2 -8137.067} C_VEL
LIN {X 0,Y 460.548,Z 441.743,A -85,B 0,C 180,E1 -8140.269,E2 -8140.269} C_VEL
LIN {X 0,Y 460.514,Z 441.748,A -85,B 0,C 180,E1 -8143.374,E2 -8143.374} C_VEL
LIN {X 0,Y 460.505,Z 441.752,A -85,B 0,C 180,E1 -8146.624,E2 -8146.624} C_VEL
LIN {X 0,Y 460.568,Z 441.743,A -85,B 0,C 180,E1 -8149.727,E2 -8149.727} C_VEL
LIN {X 0,Y 460.625,Z 441.833,A -85,B 0,C 180,E1 -8150.39,E2 -8150.39} C_VEL
LIN {X 0,Y 461.107,Z 446.753,A -85,B 0,C 180,E1 -8152.434,E2 -8152.434} C_VEL
LIN {X 0,Y 460.925,Z 454.556,A -85,B 0,C 180,E1 -8155.655,E2 -8155.655} C_VEL
LIN {X 0,Y 460.755,Z 462.072,A -85,B 0,C 180,E1 -8158.76,E2 -8158.76} C_VEL
LIN {X 0,Y 460.618,Z 469.338,A -85,B 0,C 180,E1 -8161.77,E2 -8161.77} C_VEL
LIN {X 0,Y 460.436,Z 476.511,A -85,B 0,C 180,E1 -8164.697,E2 -8164.697} C_VEL
LIN {X 0,Y 460.286,Z 484.89,A -85,B 0,C 180,E1 -8168.031,E2 -8168.031} C_VEL
LIN {X 0,Y 460.21,Z 490.067,A -85,B 0,C 180,E1 -8170.029,E2 -8170.029} C_VEL
LIN {X 0,Y 460.103,Z 491.909,A -85,B 0,C 180,E1 -8170.438,E2 -8170.438} C_VEL
LIN {X 0,Y 459.897,Z 494.664,A -85,B 0,C 180,E1 -8170.765,E2 -8170.765} C_VEL
LIN {X 0,Y 459.479,Z 499.79,A -85,B 0,C 180,E1 -8171.122,E2 -8171.122} C_VEL
LIN {X 0,Y 458.995,Z 505.975,A -85,B 0,C 180,E1 -8171.36,E2 -8171.36} C_VEL
LIN {X 0,Y 458.272,Z 518.235,A -85,B 0,C 180,E1 -8171.752,E2 -8171.752} C_VEL
LIN {X 0,Y 457.699,Z 531.308,A -85,B 0,C 180,E1 -8172.336,E2 -8172.336} C_VEL
LIN {X 0,Y 457.04,Z 544.693,A -85,B 0,C 180,E1 -8173.126,E2 -8173.126} C_VEL
LIN {X 0,Y 456.315,Z 556.673,A -85,B 0,C 180,E1 -8174.019,E2 -8174.019} C_VEL
LIN {X 0,Y 455.612,Z 567.699,A -85,B 0,C 180,E1 -8175.025,E2 -8175.025} C_VEL
LIN {X 0,Y 454.874,Z 577.873,A -85,B 0,C 180,E1 -8176.143,E2 -8176.143} C_VEL
LIN {X 0,Y 454.258,Z 588.015,A -85,B 0,C 180,E1 -8177.49,E2 -8177.49} C_VEL
LIN {X 0,Y 453.696,Z 596.391,A -85,B 0,C 180,E1 -8178.834,E2 -8178.834} C_VEL
LIN {X 0,Y 453.188,Z 604.39,A -85,B 0,C 180,E1 -8180.402,E2 -8180.402} C_VEL
LIN {X 0,Y 452.871,Z 610.828,A -85,B 0,C 180,E1 -8181.97,E2 -8181.97} C_VEL
LIN {X 0,Y 452.653,Z 616.528,A -85,B 0,C 180,E1 -8183.759,E2 -8183.759} C_VEL
LIN {X 0,Y 452.622,Z 618.786,A -85,B 0,C 180,E1 -8184.653,E2 -8184.653} C_VEL
LIN {X 0,Y 452.479,Z 622.207,A -85,B 0,C 180,E1 -8186.437,E2 -8186.437} C_VEL
LIN {X 0,Y 452.432,Z 624.246,A -85,B 0,C 180,E1 -8188.219,E2 -8188.219} C_VEL
LIN {X 0,Y 452.406,Z 624.952,A -85,B 0,C 180,E1 -8189.999,E2 -8189.999} C_VEL
LIN {X 0,Y 452.43,Z 624.327,A -85,B 0,C 180,E1 -8191.779,E2 -8191.779} C_VEL
LIN {X 0,Y 452.478,Z 622.36,A -85,B 0,C 180,E1 -8193.561,E2 -8193.561} C_VEL
LIN {X 0,Y 452.62,Z 619.007,A -85,B 0,C 180,E1 -8195.344,E2 -8195.344} C_VEL
LIN {X 0,Y 452.714,Z 614.171,A -85,B 0,C 180,E1 -8197.133,E2 -8197.133} C_VEL
LIN {X 0,Y 453.019,Z 607.71,A -85,B 0,C 180,E1 -8198.924,E2 -8198.924} C_VEL
LIN {X 0,Y 453.396,Z 600.509,A -85,B 0,C 180,E1 -8200.493,E2 -8200.493} C_VEL
LIN {X 0,Y 454.051,Z 591.543,A -85,B 0,C 180,E1 -8202.06,E2 -8202.06} C_VEL
LIN {X 0,Y 454.546,Z 582.165,A -85,B 0,C 180,E1 -8203.409,E2 -8203.409} C_VEL
LIN {X 0,Y 455.338,Z 571.782,A -85,B 0,C 180,E1 -8204.639,E2 -8204.639} C_VEL
LIN {X 0,Y 456.045,Z 560.334,A -85,B 0,C 180,E1 -8205.759,E2 -8205.759} C_VEL
LIN {X 0,Y 456.88,Z 547.653,A -85,B 0,C 180,E1 -8206.762,E2 -8206.762} C_VEL
LIN {X 0,Y 457.548,Z 534.893,A -85,B 0,C 180,E1 -8207.566,E2 -8207.566} C_VEL
LIN {X 0,Y 458.128,Z 520.844,A -85,B 0,C 180,E1 -8208.24,E2 -8208.24} C_VEL
LIN {X 0,Y 458.105,Z 516.184,A -85,B 0,C 180,E1 -8208.428,E2 -8208.428} C_VEL
LIN {X 0,Y 455.25,Z 501.972,A -85,B 0,C 180,E1 -8208.993,E2 -8208.993} C_VEL
LIN {X 0,Y 453.118,Z 492.967,A -85,B 0,C 180,E1 -8209.273,E2 -8209.273} C_VEL
LIN {X 0,Y 453.268,Z 486.293,A -85,B 0,C 180,E1 -8211.845,E2 -8211.845} C_VEL
LIN {X 0,Y 453.411,Z 477.803,A -85,B 0,C 180,E1 -8215.229,E2 -8215.229} C_VEL
LIN {X 0,Y 453.593,Z 471.12,A -85,B 0,C 180,E1 -8217.973,E2 -8217.973} C_VEL
LIN {X 0,Y 453.717,Z 464.53,A -85,B 0,C 180,E1 -8220.74,E2 -8220.74} C_VEL
LIN {X 0,Y 453.95,Z 455.864,A -85,B 0,C 180,E1 -8224.363,E2 -8224.363} C_VEL
LIN {X 0,Y 454.113,Z 447.429,A -85,B 0,C 180,E1 -8227.88,E2 -8227.88} C_VEL
LIN {X 0,Y 453.575,Z 442.635,A -85,B 0,C 180,E1 -8229.889,E2 -8229.889} C_VEL
LIN {X 0,Y 453.476,Z 442.624,A -85,B 0,C 180,E1 -8233.247,E2 -8233.247} C_VEL
LIN {X 0,Y 453.47,Z 442.626,A -85,B 0,C 180,E1 -8235.779,E2 -8235.779} C_VEL
LIN {X 0,Y 453.489,Z 442.624,A -85,B 0,C 180,E1 -8238.21,E2 -8238.21} C_VEL
LIN {X 0,Y 453.523,Z 442.616,A -85,B 0,C 180,E1 -8240.787,E2 -8240.787} C_VEL
LIN {X 0,Y 453.449,Z 442.625,A -85,B 0,C 180,E1 -8243.916,E2 -8243.916} C_VEL
LIN {X 0,Y 453.474,Z 442.623,A -85,B 0,C 180,E1 -8247.15,E2 -8247.15} C_VEL
LIN {X 0,Y 453.505,Z 442.622,A -85,B 0,C 180,E1 -8250.27,E2 -8250.27} C_VEL
LIN {X 0,Y 453.504,Z 442.616,A -85,B 0,C 180,E1 -8253.294,E2 -8253.294} C_VEL
LIN {X 0,Y 453.495,Z 442.619,A -85,B 0,C 180,E1 -8256.238,E2 -8256.238} C_VEL
LIN {X 0,Y 453.498,Z 442.618,A -85,B 0,C 180,E1 -8259.118,E2 -8259.118} C_VEL
LIN {X 0,Y 453.502,Z 442.621,A -85,B 0,C 180,E1 -8261.944,E2 -8261.944} C_VEL
LIN {X 0,Y 453.539,Z 442.612,A -85,B 0,C 180,E1 -8264.726,E2 -8264.726} C_VEL
LIN {X 0,Y 453.591,Z 442.608,A -85,B 0,C 180,E1 -8267.472,E2 -8267.472} C_VEL
LIN {X 0,Y 453.584,Z 442.608,A -85,B 0,C 180,E1 -8271.086,E2 -8271.086} C_VEL
LIN {X 0,Y 453.674,Z 442.598,A -85,B 0,C 180,E1 -8273.775,E2 -8273.775} C_VEL
LIN {X 0,Y 453.757,Z 442.588,A -85,B 0,C 180,E1 -8277.337,E2 -8277.337} C_VEL
LIN {X 0,Y 453.813,Z 442.58,A -85,B 0,C 180,E1 -8280,E2 -8280} C_VEL
LIN {X 0,Y 453.756,Z 442.582,A -85,B 0,C 180,E1 -8282.663,E2 -8282.663} C_VEL
LIN {X 0,Y 453.667,Z 442.599,A -85,B 0,C 180,E1 -8286.225,E2 -8286.225} C_VEL
LIN {X 0,Y 453.583,Z 442.604,A -85,B 0,C 180,E1 -8288.913,E2 -8288.913} C_VEL
LIN {X 0,Y 453.59,Z 442.604,A -85,B 0,C 180,E1 -8292.551,E2 -8292.551} C_VEL
LIN {X 0,Y 453.533,Z 442.611,A -85,B 0,C 180,E1 -8296.196,E2 -8296.196} C_VEL
LIN {X 0,Y 453.51,Z 442.616,A -85,B 0,C 180,E1 -8299.041,E2 -8299.041} C_VEL
LIN {X 0,Y 453.467,Z 442.626,A -85,B 0,C 180,E1 -8301.837,E2 -8301.837} C_VEL
LIN {X 0,Y 453.504,Z 442.617,A -85,B 0,C 180,E1 -8304.735,E2 -8304.735} C_VEL
LIN {X 0,Y 453.529,Z 442.613,A -85,B 0,C 180,E1 -8307.962,E2 -8307.962} C_VEL
LIN {X 0,Y 453.474,Z 442.624,A -85,B 0,C 180,E1 -8310.76,E2 -8310.76} C_VEL
LIN {X 0,Y 453.469,Z 442.625,A -85,B 0,C 180,E1 -8313.913,E2 -8313.913} C_VEL
LIN {X 0,Y 453.463,Z 442.624,A -85,B 0,C 180,E1 -8317.189,E2 -8317.189} C_VEL
LIN {X 0,Y 453.525,Z 442.62,A -85,B 0,C 180,E1 -8319.446,E2 -8319.446} C_VEL
LIN {X 0,Y 453.485,Z 442.624,A -85,B 0,C 180,E1 -8322.992,E2 -8322.992} C_VEL
LIN {X 0,Y 453.459,Z 442.626,A -85,B 0,C 180,E1 -8325.78,E2 -8325.78} C_VEL
LIN {X 0,Y 453.51,Z 442.621,A -85,B 0,C 180,E1 -8329.407,E2 -8329.407} C_VEL
LIN {X 0,Y 453.5,Z 442.684,A -85,B 0,C 180,E1 -8331.842,E2 -8331.842} C_VEL
LIN {X 0,Y 455.15,Z 451.346,A -85,B 0,C 180,E1 -8335.159,E2 -8335.159} C_VEL
LIN {X 0,Y 455.978,Z 456.006,A -85,B 0,C 180,E1 -8336.871,E2 -8336.871} C_VEL
LIN {X 0,Y 455.679,Z 461.917,A -85,B 0,C 180,E1 -8338.892,E2 -8338.892} C_VEL
LIN {X 0,Y 455.017,Z 471.384,A -85,B 0,C 180,E1 -8342.034,E2 -8342.034} C_VEL
LIN {X 0,Y 454.494,Z 480.049,A -85,B 0,C 180,E1 -8344.835,E2 -8344.835} C_VEL
LIN {X 0,Y 453.927,Z 490.687,A -85,B 0,C 180,E1 -8348.188,E2 -8348.188} C_VEL
LIN {X 0,Y 453.542,Z 499.916,A -85,B 0,C 180,E1 -8351.028,E2 -8351.028} C_VEL
LIN {X 0,Y 456.579,Z 516.373,A -85,B 0,C 180,E1 -8351.544,E2 -8351.544} C_VEL
LIN {X 0,Y 457.669,Z 524.217,A -85,B 0,C 180,E1 -8351.855,E2 -8351.855} C_VEL
LIN {X 0,Y 457.145,Z 538.417,A -85,B 0,C 180,E1 -8352.468,E2 -8352.468} C_VEL
LIN {X 0,Y 456.55,Z 551.537,A -85,B 0,C 180,E1 -8353.225,E2 -8353.225} C_VEL
LIN {X 0,Y 455.812,Z 563.764,A -85,B 0,C 180,E1 -8354.118,E2 -8354.118} C_VEL
LIN {X 0,Y 455.095,Z 574.941,A -85,B 0,C 180,E1 -8355.125,E2 -8355.125} C_VEL
LIN {X 0,Y 454.428,Z 586.135,A -85,B 0,C 180,E1 -8356.36,E2 -8356.36} C_VEL
LIN {X 0,Y 453.865,Z 596.133,A -85,B 0,C 180,E1 -8357.708,E2 -8357.708} C_VEL
LIN {X 0,Y 453.402,Z 604.414,A -85,B 0,C 180,E1 -8359.055,E2 -8359.055} C_VEL
LIN {X 0,Y 452.993,Z 612.309,A -85,B 0,C 180,E1 -8360.626,E2 -8360.626} C_VEL
LIN {X 0,Y 452.729,Z 617.83,A -85,B 0,C 180,E1 -8361.97,E2 -8361.97} C_VEL
LIN {X 0,Y 452.602,Z 623.604,A -85,B 0,C 180,E1 -8363.761,E2 -8363.761} C_VEL
LIN {X 0,Y 452.582,Z 625.889,A -85,B 0,C 180,E1 -8364.655,E2 -8364.655} C_VEL
LIN {X 0,Y 452.503,Z 629.338,A -85,B 0,C 180,E1 -8366.439,E2 -8366.439} C_VEL
LIN {X 0,Y 452.476,Z 631.376,A -85,B 0,C 180,E1 -8368.221,E2 -8368.221} C_VEL
LIN {X 0,Y 452.433,Z 632.053,A -85,B 0,C 180,E1 -8370.001,E2 -8370.001} C_VEL
LIN {X 0,Y 452.488,Z 631.373,A -85,B 0,C 180,E1 -8371.781,E2 -8371.781} C_VEL
LIN {X 0,Y 452.502,Z 629.33,A -85,B 0,C 180,E1 -8373.563,E2 -8373.563} C_VEL
LIN {X 0,Y 452.584,Z 625.881,A -85,B 0,C 180,E1 -8375.347,E2 -8375.347} C_VEL
LIN {X 0,Y 452.658,Z 620.918,A -85,B 0,C 180,E1 -8377.136,E2 -8377.136} C_VEL
LIN {X 0,Y 452.914,Z 614.287,A -85,B 0,C 180,E1 -8378.928,E2 -8378.928} C_VEL
LIN {X 0,Y 453.242,Z 606.859,A -85,B 0,C 180,E1 -8380.499,E2 -8380.499} C_VEL
LIN {X 0,Y 453.719,Z 599.08,A -85,B 0,C 180,E1 -8381.845,E2 -8381.845} C_VEL
LIN {X 0,Y 454.222,Z 589.546,A -85,B 0,C 180,E1 -8383.209,E2 -8383.209} C_VEL
LIN {X 0,Y 454.907,Z 579.225,A -85,B 0,C 180,E1 -8384.426,E2 -8384.426} C_VEL
LIN {X 0,Y 455.5,Z 568.95,A -85,B 0,C 180,E1 -8385.437,E2 -8385.437} C_VEL
LIN {X 0,Y 456.254,Z 556.366,A -85,B 0,C 180,E1 -8386.443,E2 -8386.443} C_VEL
LIN {X 0,Y 456.898,Z 543.942,A -85,B 0,C 180,E1 -8387.236,E2 -8387.236} C_VEL
LIN {X 0,Y 457.453,Z 530.555,A -85,B 0,C 180,E1 -8387.896,E2 -8387.896} C_VEL
LIN {X 0,Y 457.579,Z 522.616,A -85,B 0,C 180,E1 -8388.209,E2 -8388.209} C_VEL
LIN {X 0,Y 455.095,Z 506.933,A -85,B 0,C 180,E1 -8388.767,E2 -8388.767} C_VEL
LIN {X 0,Y 453.52,Z 499.066,A -85,B 0,C 180,E1 -8389.04,E2 -8389.04} C_VEL
LIN {X 0,Y 453.951,Z 488.754,A -85,B 0,C 180,E1 -8392.292,E2 -8392.292} C_VEL
LIN {X 0,Y 454.48,Z 480.107,A -85,B 0,C 180,E1 -8395.168,E2 -8395.168} C_VEL
LIN {X 0,Y 455.303,Z 471.1,A -85,B 0,C 180,E1 -8398.376,E2 -8398.376} C_VEL
LIN {X 0,Y 456.308,Z 462.986,A -85,B 0,C 180,E1 -8401.579,E2 -8401.579} C_VEL
LIN {X 0,Y 456.702,Z 459.507,A -85,B 0,C 180,E1 -8403.114,E2 -8403.114} C_VEL
LIN {X 0,Y 456.254,Z 456.392,A -85,B 0,C 180,E1 -8404.747,E2 -8404.747} C_VEL
LIN {X 0,Y 455.559,Z 452.746,A -85,B 0,C 180,E1 -8406.99,E2 -8406.99} C_VEL
LIN {X 0,Y 454.998,Z 449.661,A -85,B 0,C 180,E1 -8409.438,E2 -8409.438} C_VEL
LIN {X 0,Y 454.516,Z 447.476,A -85,B 0,C 180,E1 -8412.08,E2 -8412.08} C_VEL
LIN {X 0,Y 454.259,Z 446.499,A -85,B 0,C 180,E1 -8414.628,E2 -8414.628} C_VEL
LIN {X 0,Y 454.26,Z 446.565,A -85,B 0,C 180,E1 -8417.099,E2 -8417.099} C_VEL
LIN {X 0,Y 454.425,Z 447.498,A -85,B 0,C 180,E1 -8419.492,E2 -8419.492} C_VEL
LIN {X 0,Y 454.722,Z 449.29,A -85,B 0,C 180,E1 -8422.022,E2 -8422.022} C_VEL
LIN {X 0,Y 454.856,Z 451.252,A -85,B 0,C 180,E1 -8424.046,E2 -8424.046} C_VEL
LIN {X 0,Y 454.603,Z 453.792,A -85,B 0,C 180,E1 -8426.183,E2 -8426.183} C_VEL
LIN {X 0,Y 454.18,Z 458.02,A -85,B 0,C 180,E1 -8429.293,E2 -8429.293} C_VEL
LIN {X 0,Y 453.828,Z 462.549,A -85,B 0,C 180,E1 -8432.317,E2 -8432.317} C_VEL
LIN {X 0,Y 453.499,Z 467.279,A -85,B 0,C 180,E1 -8435.265,E2 -8435.265} C_VEL
LIN {X 0,Y 453.294,Z 472.675,A -85,B 0,C 180,E1 -8438.477,E2 -8438.477} C_VEL
LIN {X 0,Y 453.112,Z 477.269,A -85,B 0,C 180,E1 -8441.112,E2 -8441.112} C_VEL
LIN {X 0,Y 452.971,Z 482.124,A -85,B 0,C 180,E1 -8443.814,E2 -8443.814} C_VEL
LIN {X 0,Y 456.033,Z 494.727,A -85,B 0,C 180,E1 -8444.383,E2 -8444.383} C_VEL
LIN {X 0,Y 456.965,Z 501.015,A -85,B 0,C 180,E1 -8444.701,E2 -8444.701} C_VEL
LIN {X 0,Y 456.417,Z 514.007,A -85,B 0,C 180,E1 -8445.396,E2 -8445.396} C_VEL
LIN {X 0,Y 455.878,Z 525.11,A -85,B 0,C 180,E1 -8446.157,E2 -8446.157} C_VEL
LIN {X 0,Y 455.303,Z 535.813,A -85,B 0,C 180,E1 -8447.067,E2 -8447.067} C_VEL
LIN {X 0,Y 454.65,Z 546.438,A -85,B 0,C 180,E1 -8448.181,E2 -8448.181} C_VEL
LIN {X 0,Y 454.118,Z 555.177,A -85,B 0,C 180,E1 -8449.297,E2 -8449.297} C_VEL
LIN {X 0,Y 453.646,Z 563.767,A -85,B 0,C 180,E1 -8450.638,E2 -8450.638} C_VEL
LIN {X 0,Y 453.227,Z 570.648,A -85,B 0,C 180,E1 -8451.978,E2 -8451.978} C_VEL
LIN {X 0,Y 452.952,Z 575.862,A -85,B 0,C 180,E1 -8453.233,E2 -8453.233} C_VEL
LIN {X 0,Y 452.701,Z 580.499,A -85,B 0,C 180,E1 -8454.655,E2 -8454.655} C_VEL
LIN {X 0,Y 452.748,Z 582.777,A -85,B 0,C 180,E1 -8455.549,E2 -8455.549} C_VEL
LIN {X 0,Y 452.667,Z 584.635,A -85,B 0,C 180,E1 -8456.44,E2 -8456.44} C_VEL
LIN {X 0,Y 452.591,Z 586.032,A -85,B 0,C 180,E1 -8457.33,E2 -8457.33} C_VEL
LIN {X 0,Y 452.559,Z 587.011,A -85,B 0,C 180,E1 -8458.22,E2 -8458.22} C_VEL
LIN {X 0,Y 452.465,Z 587.801,A -85,B 0,C 180,E1 -8460,E2 -8460} C_VEL
LIN {X 0,Y 452.491,Z 587.563,A -85,B 0,C 180,E1 -8460.89,E2 -8460.89} C_VEL
LIN {X 0,Y 452.544,Z 586.916,A -85,B 0,C 180,E1 -8461.78,E2 -8461.78} C_VEL
LIN {X 0,Y 452.662,Z 584.439,A -85,B 0,C 180,E1 -8463.561,E2 -8463.561} C_VEL
LIN {X 0,Y 452.646,Z 581.44,A -85,B 0,C 180,E1 -8464.899,E2 -8464.899} C_VEL
LIN {X 0,Y 452.905,Z 577.388,A -85,B 0,C 180,E1 -8466.236,E2 -8466.236} C_VEL
LIN {X 0,Y 453.053,Z 571.187,A -85,B 0,C 180,E1 -8467.801,E2 -8467.801} C_VEL
LIN {X 0,Y 453.416,Z 564.421,A -85,B 0,C 180,E1 -8469.142,E2 -8469.142} C_VEL
LIN {X 0,Y 453.855,Z 556.057,A -85,B 0,C 180,E1 -8470.483,E2 -8470.483} C_VEL
LIN {X 0,Y 454.286,Z 547.519,A -85,B 0,C 180,E1 -8471.602,E2 -8471.602} C_VEL
LIN {X 0,Y 454.944,Z 537.243,A -85,B 0,C 180,E1 -8472.697,E2 -8472.697} C_VEL
LIN {X 0,Y 455.48,Z 525.374,A -85,B 0,C 180,E1 -8473.723,E2 -8473.723} C_VEL
LIN {X 0,Y 456.021,Z 513.867,A -85,B 0,C 180,E1 -8474.504,E2 -8474.504} C_VEL
LIN {X 0,Y 456.492,Z 501.049,A -85,B 0,C 180,E1 -8475.173,E2 -8475.173} C_VEL
LIN {X 0,Y 455.448,Z 493.374,A -85,B 0,C 180,E1 -8475.532,E2 -8475.532} C_VEL
LIN {X 0,Y 452.783,Z 480.742,A -85,B 0,C 180,E1 -8476.039,E2 -8476.039} C_VEL
LIN {X 0,Y 452.904,Z 475.073,A -85,B 0,C 180,E1 -8479.018,E2 -8479.018} C_VEL
LIN {X 0,Y 453.016,Z 469.748,A -85,B 0,C 180,E1 -8481.86,E2 -8481.86} C_VEL
LIN {X 0,Y 453.152,Z 464.404,A -85,B 0,C 180,E1 -8484.756,E2 -8484.756} C_VEL
LIN {X 0,Y 453.347,Z 458.674,A -85,B 0,C 180,E1 -8487.914,E2 -8487.914} C_VEL
LIN {X 0,Y 453.498,Z 453.601,A -85,B 0,C 180,E1 -8490.758,E2 -8490.758} C_VEL
LIN {X 0,Y 453.681,Z 448.118,A -85,B 0,C 180,E1 -8493.896,E2 -8493.896} C_VEL
LIN {X 0,Y 453.668,Z 443.314,A -85,B 0,C 180,E1 -8496.715,E2 -8496.715} C_VEL
LIN {X 0,Y 453.527,Z 442.62,A -85,B 0,C 180,E1 -8497.183,E2 -8497.183} C_VEL
LIN {X 0,Y 453.5,Z 442.62,A -85,B 0,C 180,E1 -8500.591,E2 -8500.591} C_VEL
LIN {X 0,Y 453.469,Z 442.626,A -85,B 0,C 180,E1 -8503.245,E2 -8503.245} C_VEL
LIN {X 0,Y 453.472,Z 442.627,A -85,B 0,C 180,E1 -8505.779,E2 -8505.779} C_VEL
LIN {X 0,Y 453.522,Z 442.621,A -85,B 0,C 180,E1 -8509.405,E2 -8509.405} C_VEL
LIN {X 0,Y 453.579,Z 442.792,A -85,B 0,C 180,E1 -8510.271,E2 -8510.271} C_VEL
LIN {X 0,Y 454.076,Z 447.168,A -85,B 0,C 180,E1 -8512.126,E2 -8512.126} C_VEL
LIN {X 0,Y 453.918,Z 454.426,A -85,B 0,C 180,E1 -8515.145,E2 -8515.145} C_VEL
LIN {X 0,Y 453.745,Z 462.265,A -85,B 0,C 180,E1 -8518.418,E2 -8518.418} C_VEL
LIN {X 0,Y 453.582,Z 469.135,A -85,B 0,C 180,E1 -8521.292,E2 -8521.292} C_VEL
LIN {X 0,Y 453.431,Z 476.366,A -85,B 0,C 180,E1 -8524.278,E2 -8524.278} C_VEL
LIN {X 0,Y 453.241,Z 484.814,A -85,B 0,C 180,E1 -8527.672,E2 -8527.672} C_VEL
LIN {X 0,Y 453.117,Z 492.181,A -85,B 0,C 180,E1 -8530.523,E2 -8530.523} C_VEL
LIN {X 0,Y 453.105,Z 492.942,A -85,B 0,C 180,E1 -8530.813,E2 -8530.813} C_VEL
LIN {X 0,Y 456.772,Z 508.966,A -85,B 0,C 180,E1 -8531.357,E2 -8531.357} C_VEL
LIN {X 0,Y 458.291,Z 517.503,A -85,B 0,C 180,E1 -8531.723,E2 -8531.723} C_VEL
LIN {X 0,Y 458.272,Z 518.235,A -85,B 0,C 180,E1 -8531.752,E2 -8531.752} C_VEL
LIN {X 0,Y 457.45,Z 523.91,A -85,B 0,C 180,E1 -8531.957,E2 -8531.957} C_VEL
LIN {X 0,Y 454.272,Z 532.934,A -85,B 0,C 180,E1 -8532.277,E2 -8532.277} C_VEL
LIN {X 0,Y 451.037,Z 541.734,A -85,B 0,C 180,E1 -8532.681,E2 -8532.681} C_VEL
LIN {X 0,Y 450.131,Z 546.931,A -85,B 0,C 180,E1 -8533.014,E2 -8533.014} C_VEL
LIN {X 0,Y 449.235,Z 559.356,A -85,B 0,C 180,E1 -8533.993,E2 -8533.993} C_VEL
LIN {X 0,Y 448.494,Z 570.981,A -85,B 0,C 180,E1 -8535.131,E2 -8535.131} C_VEL
LIN {X 0,Y 447.699,Z 581.503,A -85,B 0,C 180,E1 -8536.38,E2 -8536.38} C_VEL
LIN {X 0,Y 447.142,Z 590.999,A -85,B 0,C 180,E1 -8537.748,E2 -8537.748} C_VEL
LIN {X 0,Y 446.487,Z 598.878,A -85,B 0,C 180,E1 -8539.111,E2 -8539.111} C_VEL
LIN {X 0,Y 446.097,Z 605.437,A -85,B 0,C 180,E1 -8540.477,E2 -8540.477} C_VEL
LIN {X 0,Y 445.829,Z 610.883,A -85,B 0,C 180,E1 -8541.843,E2 -8541.843} C_VEL
LIN {X 0,Y 445.579,Z 616.584,A -85,B 0,C 180,E1 -8543.66,E2 -8543.66} C_VEL
LIN {X 0,Y 445.54,Z 618.842,A -85,B 0,C 180,E1 -8544.568,E2 -8544.568} C_VEL
LIN {X 0,Y 445.379,Z 622.263,A -85,B 0,C 180,E1 -8546.38,E2 -8546.38} C_VEL
LIN {X 0,Y 445.351,Z 624.302,A -85,B 0,C 180,E1 -8548.19,E2 -8548.19} C_VEL
LIN {X 0,Y 445.315,Z 625.007,A -85,B 0,C 180,E1 -8549.999,E2 -8549.999} C_VEL
LIN {X 0,Y 445.35,Z 624.383,A -85,B 0,C 180,E1 -8551.807,E2 -8551.807} C_VEL
LIN {X 0,Y 445.378,Z 622.414,A -85,B 0,C 180,E1 -8553.618,E2 -8553.618} C_VEL
LIN {X 0,Y 445.539,Z 619.06,A -85,B 0,C 180,E1 -8555.43,E2 -8555.43} C_VEL
LIN {X 0,Y 445.659,Z 614.223,A -85,B 0,C 180,E1 -8557.246,E2 -8557.246} C_VEL
LIN {X 0,Y 445.974,Z 607.761,A -85,B 0,C 180,E1 -8559.066,E2 -8559.066} C_VEL
LIN {X 0,Y 446.376,Z 600.559,A -85,B 0,C 180,E1 -8560.66,E2 -8560.66} C_VEL
LIN {X 0,Y 447.075,Z 591.591,A -85,B 0,C 180,E1 -8562.251,E2 -8562.251} C_VEL
LIN {X 0,Y 447.605,Z 582.211,A -85,B 0,C 180,E1 -8563.621,E2 -8563.621} C_VEL
LIN {X 0,Y 448.45,Z 571.824,A -85,B 0,C 180,E1 -8564.869,E2 -8564.869} C_VEL
LIN {X 0,Y 449.203,Z 560.372,A -85,B 0,C 180,E1 -8566.005,E2 -8566.005} C_VEL
LIN {X 0,Y 450.078,Z 547.685,A -85,B 0,C 180,E1 -8567.023,E2 -8567.023} C_VEL
LIN {X 0,Y 450.797,Z 534.682,A -85,B 0,C 180,E1 -8567.852,E2 -8567.852} C_VEL
LIN {X 0,Y 451.422,Z 520.407,A -85,B 0,C 180,E1 -8568.539,E2 -8568.539} C_VEL
LIN {X 0,Y 451.243,Z 516.811,A -85,B 0,C 180,E1 -8568.693,E2 -8568.693} C_VEL
LIN {X 0,Y 448.425,Z 502.591,A -85,B 0,C 180,E1 -8569.277,E2 -8569.277} C_VEL
LIN {X 0,Y 446.053,Z 492.937,A -85,B 0,C 180,E1 -8569.599,E2 -8569.599} C_VEL
LIN {X 0,Y 446.208,Z 486.225,A -85,B 0,C 180,E1 -8572.209,E2 -8572.209} C_VEL
LIN {X 0,Y 446.376,Z 477.671,A -85,B 0,C 180,E1 -8575.655,E2 -8575.655} C_VEL
LIN {X 0,Y 446.553,Z 470.395,A -85,B 0,C 180,E1 -8578.685,E2 -8578.685} C_VEL
LIN {X 0,Y 446.686,Z 464.278,A -85,B 0,C 180,E1 -8581.278,E2 -8581.278} C_VEL
LIN {X 0,Y 446.95,Z 456.703,A -85,B 0,C 180,E1 -8584.475,E2 -8584.475} C_VEL
LIN {X 0,Y 447.116,Z 448.808,A -85,B 0,C 180,E1 -8587.806,E2 -8587.806} C_VEL
LIN {X 0,Y 446.754,Z 444.64,A -85,B 0,C 180,E1 -8589.571,E2 -8589.571} C_VEL
LIN {X 0,Y 446.517,Z 443.493,A -85,B 0,C 180,E1 -8590.094,E2 -8590.094} C_VEL
LIN {X 0,Y 446.441,Z 443.5,A -85,B 0,C 180,E1 -8593.602,E2 -8593.602} C_VEL
LIN {X 0,Y 446.44,Z 443.503,A -85,B 0,C 180,E1 -8596.396,E2 -8596.396} C_VEL
LIN {X 0,Y 446.461,Z 443.497,A -85,B 0,C 180,E1 -8599.804,E2 -8599.804} C_VEL
LIN {X 0,Y 446.425,Z 443.499,A -85,B 0,C 180,E1 -8602.123,E2 -8602.123} C_VEL
LIN {X 0,Y 446.422,Z 443.497,A -85,B 0,C 180,E1 -8605.476,E2 -8605.476} C_VEL
LIN {X 0,Y 446.411,Z 443.498,A -85,B 0,C 180,E1 -8608.699,E2 -8608.699} C_VEL
LIN {X 0,Y 446.475,Z 443.496,A -85,B 0,C 180,E1 -8611.821,E2 -8611.821} C_VEL
LIN {X 0,Y 446.449,Z 443.497,A -85,B 0,C 180,E1 -8614.847,E2 -8614.847} C_VEL
LIN {X 0,Y 446.461,Z 443.489,A -85,B 0,C 180,E1 -8618.237,E2 -8618.237} C_VEL
LIN {X 0,Y 446.448,Z 443.498,A -85,B 0,C 180,E1 -8621.649,E2 -8621.649} C_VEL
LIN {X 0,Y 446.506,Z 443.489,A -85,B 0,C 180,E1 -8624.48,E2 -8624.48} C_VEL
LIN {X 0,Y 446.53,Z 443.484,A -85,B 0,C 180,E1 -8628.193,E2 -8628.193} C_VEL
LIN {X 0,Y 446.589,Z 443.477,A -85,B 0,C 180,E1 -8631.858,E2 -8631.858} C_VEL
LIN {X 0,Y 446.644,Z 443.472,A -85,B 0,C 180,E1 -8634.583,E2 -8634.583} C_VEL
LIN {X 0,Y 446.701,Z 443.467,A -85,B 0,C 180,E1 -8637.295,E2 -8637.295} C_VEL
LIN {X 0,Y 446.784,Z 443.456,A -85,B 0,C 180,E1 -8640,E2 -8640} C_VEL
LIN {X 0,Y 446.7,Z 443.46,A -85,B 0,C 180,E1 -8642.705,E2 -8642.705} C_VEL
LIN {X 0,Y 446.636,Z 443.476,A -85,B 0,C 180,E1 -8646.324,E2 -8646.324} C_VEL
LIN {X 0,Y 446.529,Z 443.483,A -85,B 0,C 180,E1 -8649.055,E2 -8649.055} C_VEL
LIN {X 0,Y 446.523,Z 443.485,A -85,B 0,C 180,E1 -8652.73,E2 -8652.73} C_VEL
LIN {X 0,Y 446.479,Z 443.49,A -85,B 0,C 180,E1 -8656.459,E2 -8656.459} C_VEL
LIN {X 0,Y 446.459,Z 443.493,A -85,B 0,C 180,E1 -8659.304,E2 -8659.304} C_VEL
LIN {X 0,Y 446.409,Z 443.503,A -85,B 0,C 180,E1 -8662.2,E2 -8662.2} C_VEL
LIN {X 0,Y 446.448,Z 443.499,A -85,B 0,C 180,E1 -8665.153,E2 -8665.153} C_VEL
LIN {X 0,Y 446.474,Z 443.492,A -85,B 0,C 180,E1 -8668.179,E2 -8668.179} C_VEL
LIN {X 0,Y 446.41,Z 443.501,A -85,B 0,C 180,E1 -8671.301,E2 -8671.301} C_VEL
LIN {X 0,Y 446.422,Z 443.502,A -85,B 0,C 180,E1 -8674.524,E2 -8674.524} C_VEL
LIN {X 0,Y 446.43,Z 443.5,A -85,B 0,C 180,E1 -8678.084,E2 -8678.084} C_VEL
LIN {X 0,Y 446.44,Z 443.502,A -85,B 0,C 180,E1 -8680.922,E2 -8680.922} C_VEL
LIN {X 0,Y 446.438,Z 443.499,A -85,B 0,C 180,E1 -8683.841,E2 -8683.841} C_VEL
LIN {X 0,Y 446.392,Z 443.508,A -85,B 0,C 180,E1 -8686.404,E2 -8686.404} C_VEL
LIN {X 0,Y 446.462,Z 443.499,A -85,B 0,C 180,E1 -8689.806,E2 -8689.806} C_VEL
LIN {X 0,Y 446.479,Z 443.576,A -85,B 0,C 180,E1 -8691.545,E2 -8691.545} C_VEL
LIN {X 0,Y 447.979,Z 451.589,A -85,B 0,C 180,E1 -8694.665,E2 -8694.665} C_VEL
LIN {X 0,Y 448.996,Z 457.228,A -85,B 0,C 180,E1 -8696.782,E2 -8696.782} C_VEL
LIN {X 0,Y 448.816,Z 461.744,A -85,B 0,C 180,E1 -8698.362,E2 -8698.362} C_VEL
LIN {X 0,Y 448.119,Z 470.82,A -85,B 0,C 180,E1 -8701.434,E2 -8701.434} C_VEL
LIN {X 0,Y 447.536,Z 479.862,A -85,B 0,C 180,E1 -8704.416,E2 -8704.416} C_VEL
LIN {X 0,Y 447.009,Z 488.943,A -85,B 0,C 180,E1 -8707.346,E2 -8707.346} C_VEL
LIN {X 0,Y 446.537,Z 499.664,A -85,B 0,C 180,E1 -8710.725,E2 -8710.725} C_VEL
LIN {X 0,Y 449.418,Z 514.954,A -85,B 0,C 180,E1 -8711.194,E2 -8711.194} C_VEL
LIN {X 0,Y 450.869,Z 525.328,A -85,B 0,C 180,E1 -8711.615,E2 -8711.615} C_VEL
LIN {X 0,Y 450.319,Z 539.294,A -85,B 0,C 180,E1 -8712.241,E2 -8712.241} C_VEL
LIN {X 0,Y 449.753,Z 551.504,A -85,B 0,C 180,E1 -8712.964,E2 -8712.964} C_VEL
LIN {X 0,Y 448.965,Z 563.725,A -85,B 0,C 180,E1 -8713.869,E2 -8713.869} C_VEL
LIN {X 0,Y 448.203,Z 574.898,A -85,B 0,C 180,E1 -8714.891,E2 -8714.891} C_VEL
LIN {X 0,Y 447.49,Z 586.088,A -85,B 0,C 180,E1 -8716.144,E2 -8716.144} C_VEL
LIN {X 0,Y 446.863,Z 596.084,A -85,B 0,C 180,E1 -8717.512,E2 -8717.512} C_VEL
LIN {X 0,Y 446.411,Z 604.363,A -85,B 0,C 180,E1 -8718.882,E2 -8718.882} C_VEL
LIN {X 0,Y 445.944,Z 612.257,A -85,B 0,C 180,E1 -8720.476,E2 -8720.476} C_VEL
LIN {X 0,Y 445.675,Z 617.777,A -85,B 0,C 180,E1 -8721.842,E2 -8721.842} C_VEL
LIN {X 0,Y 445.528,Z 623.55,A -85,B 0,C 180,E1 -8723.662,E2 -8723.662} C_VEL
LIN {X 0,Y 445.403,Z 627.741,A -85,B 0,C 180,E1 -8725.476,E2 -8725.476} C_VEL
LIN {X 0,Y 445.435,Z 630.474,A -85,B 0,C 180,E1 -8727.288,E2 -8727.288} C_VEL
LIN {X 0,Y 445.365,Z 631.829,A -85,B 0,C 180,E1 -8729.097,E2 -8729.097} C_VEL
LIN {X 0,Y 445.366,Z 631.827,A -85,B 0,C 180,E1 -8730.905,E2 -8730.905} C_VEL
LIN {X 0,Y 445.436,Z 630.468,A -85,B 0,C 180,E1 -8732.714,E2 -8732.714} C_VEL
LIN {X 0,Y 445.406,Z 627.731,A -85,B 0,C 180,E1 -8734.526,E2 -8734.526} C_VEL
LIN {X 0,Y 445.53,Z 623.542,A -85,B 0,C 180,E1 -8736.341,E2 -8736.341} C_VEL
LIN {X 0,Y 445.68,Z 617.768,A -85,B 0,C 180,E1 -8738.16,E2 -8738.16} C_VEL
LIN {X 0,Y 446.024,Z 611.235,A -85,B 0,C 180,E1 -8739.753,E2 -8739.753} C_VEL
LIN {X 0,Y 446.486,Z 603.099,A -85,B 0,C 180,E1 -8741.349,E2 -8741.349} C_VEL
LIN {X 0,Y 446.959,Z 594.553,A -85,B 0,C 180,E1 -8742.718,E2 -8742.718} C_VEL
LIN {X 0,Y 447.635,Z 584.165,A -85,B 0,C 180,E1 -8744.086,E2 -8744.086} C_VEL
LIN {X 0,Y 448.33,Z 573.689,A -85,B 0,C 180,E1 -8745.224,E2 -8745.224} C_VEL
LIN {X 0,Y 449.08,Z 562.252,A -85,B 0,C 180,E1 -8746.246,E2 -8746.246} C_VEL
LIN {X 0,Y 449.802,Z 549.682,A -85,B 0,C 180,E1 -8747.153,E2 -8747.153} C_VEL
LIN {X 0,Y 450.483,Z 536.221,A -85,B 0,C 180,E1 -8747.912,E2 -8747.912} C_VEL
LIN {X 0,Y 450.822,Z 523.944,A -85,B 0,C 180,E1 -8748.439,E2 -8748.439} C_VEL
LIN {X 0,Y 448.465,Z 508.507,A -85,B 0,C 180,E1 -8749.019,E2 -8749.019} C_VEL
LIN {X 0,Y 446.529,Z 498.87,A -85,B 0,C 180,E1 -8749.379,E2 -8749.379} C_VEL
LIN {X 0,Y 447.006,Z 488.754,A -85,B 0,C 180,E1 -8752.657,E2 -8752.657} C_VEL
LIN {X 0,Y 447.556,Z 480.217,A -85,B 0,C 180,E1 -8755.585,E2 -8755.585} C_VEL
LIN {X 0,Y 448.403,Z 471.939,A -85,B 0,C 180,E1 -8758.632,E2 -8758.632} C_VEL
LIN {X 0,Y 449.391,Z 464.646,A -85,B 0,C 180,E1 -8761.595,E2 -8761.595} C_VEL
LIN {X 0,Y 449.826,Z 461.214,A -85,B 0,C 180,E1 -8763.151,E2 -8763.151} C_VEL
LIN {X 0,Y 449.199,Z 457.187,A -85,B 0,C 180,E1 -8765.373,E2 -8765.373} C_VEL
LIN {X 0,Y 448.564,Z 453.769,A -85,B 0,C 180,E1 -8767.666,E2 -8767.666} C_VEL
LIN {X 0,Y 448.069,Z 451.096,A -85,B 0,C 180,E1 -8770.024,E2 -8770.024} C_VEL
LIN {X 0,Y 447.672,Z 449.301,A -85,B 0,C 180,E1 -8772.46,E2 -8772.46} C_VEL
LIN {X 0,Y 447.445,Z 448.465,A -85,B 0,C 180,E1 -8775.024,E2 -8775.024} C_VEL
LIN {X 0,Y 447.479,Z 448.633,A -85,B 0,C 180,E1 -8777.577,E2 -8777.577} C_VEL
LIN {X 0,Y 447.639,Z 449.831,A -85,B 0,C 180,E1 -8780.293,E2 -8780.293} C_VEL
LIN {X 0,Y 447.853,Z 451.256,A -85,B 0,C 180,E1 -8782.265,E2 -8782.265} C_VEL
LIN {X 0,Y 447.925,Z 453.409,A -85,B 0,C 180,E1 -8784.512,E2 -8784.512} C_VEL
LIN {X 0,Y 447.586,Z 455.95,A -85,B 0,C 180,E1 -8786.662,E2 -8786.662} C_VEL
LIN {X 0,Y 447.147,Z 460.184,A -85,B 0,C 180,E1 -8789.822,E2 -8789.822} C_VEL
LIN {X 0,Y 446.747,Z 464.673,A -85,B 0,C 180,E1 -8792.857,E2 -8792.857} C_VEL
LIN {X 0,Y 446.453,Z 469.529,A -85,B 0,C 180,E1 -8795.929,E2 -8795.929} C_VEL
LIN {X 0,Y 446.251,Z 474.219,A -85,B 0,C 180,E1 -8798.763,E2 -8798.763} C_VEL
LIN {X 0,Y 446.033,Z 479.149,A -85,B 0,C 180,E1 -8801.631,E2 -8801.631} C_VEL
LIN {X 0,Y 445.925,Z 482.37,A -85,B 0,C 180,E1 -8803.461,E2 -8803.461} C_VEL
LIN {X 0,Y 448.97,Z 494.513,A -85,B 0,C 180,E1 -8804.046,E2 -8804.046} C_VEL
LIN {X 0,Y 450.227,Z 501.785,A -85,B 0,C 180,E1 -8804.439,E2 -8804.439} C_VEL
LIN {X 0,Y 449.623,Z 515.042,A -85,B 0,C 180,E1 -8805.17,E2 -8805.17} C_VEL
LIN {X 0,Y 449.042,Z 526.079,A -85,B 0,C 180,E1 -8805.949,E2 -8805.949} C_VEL
LIN {X 0,Y 448.424,Z 536.552,A -85,B 0,C 180,E1 -8806.865,E2 -8806.865} C_VEL
LIN {X 0,Y 447.738,Z 547.065,A -85,B 0,C 180,E1 -8807.996,E2 -8807.996} C_VEL
LIN {X 0,Y 447.173,Z 555.714,A -85,B 0,C 180,E1 -8809.129,E2 -8809.129} C_VEL
LIN {X 0,Y 446.668,Z 564.228,A -85,B 0,C 180,E1 -8810.491,E2 -8810.491} C_VEL
LIN {X 0,Y 446.223,Z 571.091,A -85,B 0,C 180,E1 -8811.851,E2 -8811.851} C_VEL
LIN {X 0,Y 445.897,Z 576.589,A -85,B 0,C 180,E1 -8813.209,E2 -8813.209} C_VEL
LIN {X 0,Y 445.655,Z 580.919,A -85,B 0,C 180,E1 -8814.571,E2 -8814.571} C_VEL
LIN {X 0,Y 445.675,Z 583.192,A -85,B 0,C 180,E1 -8815.478,E2 -8815.478} C_VEL
LIN {X 0,Y 445.609,Z 585.04,A -85,B 0,C 180,E1 -8816.383,E2 -8816.383} C_VEL
LIN {X 0,Y 445.517,Z 586.424,A -85,B 0,C 180,E1 -8817.288,E2 -8817.288} C_VEL
LIN {X 0,Y 445.471,Z 587.393,A -85,B 0,C 180,E1 -8818.192,E2 -8818.192} C_VEL
LIN {X 0,Y 445.429,Z 587.971,A -85,B 0,C 180,E1 -8819.096,E2 -8819.096} C_VEL
LIN {X 0,Y 445.401,Z 588.155,A -85,B 0,C 180,E1 -8820,E2 -8820} C_VEL
LIN {X 0,Y 445.412,Z 587.901,A -85,B 0,C 180,E1 -8820.904,E2 -8820.904} C_VEL
LIN {X 0,Y 445.457,Z 587.243,A -85,B 0,C 180,E1 -8821.808,E2 -8821.808} C_VEL
LIN {X 0,Y 445.507,Z 586.194,A -85,B 0,C 180,E1 -8822.713,E2 -8822.713} C_VEL
LIN {X 0,Y 445.601,Z 584.739,A -85,B 0,C 180,E1 -8823.617,E2 -8823.617} C_VEL
LIN {X 0,Y 445.575,Z 581.718,A -85,B 0,C 180,E1 -8824.977,E2 -8824.977} C_VEL
LIN {X 0,Y 445.827,Z 577.643,A -85,B 0,C 180,E1 -8826.335,E2 -8826.335} C_VEL
LIN {X 0,Y 446.027,Z 571.399,A -85,B 0,C 180,E1 -8827.925,E2 -8827.925} C_VEL
LIN {X 0,Y 446.412,Z 564.604,A -85,B 0,C 180,E1 -8829.286,E2 -8829.286} C_VEL
LIN {X 0,Y 446.87,Z 556.21,A -85,B 0,C 180,E1 -8830.649,E2 -8830.649} C_VEL
LIN {X 0,Y 447.34,Z 547.629,A -85,B 0,C 180,E1 -8831.785,E2 -8831.785} C_VEL
LIN {X 0,Y 448.053,Z 536.456,A -85,B 0,C 180,E1 -8832.981,E2 -8832.981} C_VEL
LIN {X 0,Y 448.585,Z 525.422,A -85,B 0,C 180,E1 -8833.938,E2 -8833.938} C_VEL
LIN {X 0,Y 449.149,Z 513.877,A -85,B 0,C 180,E1 -8834.73,E2 -8834.73} C_VEL
LIN {X 0,Y 449.617,Z 501.052,A -85,B 0,C 180,E1 -8835.41,E2 -8835.41} C_VEL
LIN {X 0,Y 447.534,Z 489.529,A -85,B 0,C 180,E1 -8835.945,E2 -8835.945} C_VEL
LIN {X 0,Y 445.732,Z 480.903,A -85,B 0,C 180,E1 -8836.27,E2 -8836.27} C_VEL
LIN {X 0,Y 445.837,Z 475.175,A -85,B 0,C 180,E1 -8839.332,E2 -8839.332} C_VEL
LIN {X 0,Y 445.965,Z 469.819,A -85,B 0,C 180,E1 -8842.223,E2 -8842.223} C_VEL
LIN {X 0,Y 446.129,Z 464.447,A -85,B 0,C 180,E1 -8845.172,E2 -8845.172} C_VEL
LIN {X 0,Y 446.311,Z 459.034,A -85,B 0,C 180,E1 -8848.191,E2 -8848.191} C_VEL
LIN {X 0,Y 446.485,Z 453.577,A -85,B 0,C 180,E1 -8851.295,E2 -8851.295} C_VEL
LIN {X 0,Y 446.666,Z 448.064,A -85,B 0,C 180,E1 -8854.502,E2 -8854.502} C_VEL
LIN {X 0,Y 446.529,Z 443.633,A -85,B 0,C 180,E1 -8857.156,E2 -8857.156} C_VEL
LIN {X 0,Y 446.454,Z 443.498,A -85,B 0,C 180,E1 -8860.197,E2 -8860.197} C_VEL
LIN {X 0,Y 446.426,Z 443.504,A -85,B 0,C 180,E1 -8863.599,E2 -8863.599} C_VEL
LIN {X 0,Y 446.405,Z 443.509,A -85,B 0,C 180,E1 -8866.403,E2 -8866.403} C_VEL
LIN {X 0,Y 446.486,Z 443.497,A -85,B 0,C 180,E1 -8869.806,E2 -8869.806} C_VEL
LIN {X 0,Y 446.556,Z 443.818,A -85,B 0,C 180,E1 -8870.166,E2 -8870.166} C_VEL
LIN {X 0,Y 447.084,Z 448.51,A -85,B 0,C 180,E1 -8872.187,E2 -8872.187} C_VEL
LIN {X 0,Y 446.922,Z 454.875,A -85,B 0,C 180,E1 -8874.857,E2 -8874.857} C_VEL
LIN {X 0,Y 446.74,Z 462.684,A -85,B 0,C 180,E1 -8878.159,E2 -8878.159} C_VEL
LIN {X 0,Y 446.6,Z 468.927,A -85,B 0,C 180,E1 -8880.8,E2 -8880.8} C_VEL
LIN {X 0,Y 446.403,Z 476.223,A -85,B 0,C 180,E1 -8883.843,E2 -8883.843} C_VEL
LIN {X 0,Y 446.232,Z 483.513,A -85,B 0,C 180,E1 -8886.812,E2 -8886.812} C_VEL
LIN {X 0,Y 446.12,Z 490.92,A -85,B 0,C 180,E1 -8889.721,E2 -8889.721} C_VEL
LIN {X 0,Y 446.078,Z 492.953,A -85,B 0,C 180,E1 -8890.503,E2 -8890.503} C_VEL
LIN {X 0,Y 449.704,Z 508.511,A -85,B 0,C 180,E1 -8891.039,E2 -8891.039} C_VEL
LIN {X 0,Y 451.533,Z 518.495,A -85,B 0,C 180,E1 -8891.479,E2 -8891.479} C_VEL
LIN {X 0,Y 450.888,Z 532.309,A -85,B 0,C 180,E1 -8892.113,E2 -8892.113} C_VEL
LIN {X 0,Y 450.249,Z 544.737,A -85,B 0,C 180,E1 -8892.864,E2 -8892.864} C_VEL
LIN {X 0,Y 450.131,Z 546.931,A -85,B 0,C 180,E1 -8893.014,E2 -8893.014} C_VEL
LIN {X 0,Y 449.242,Z 552.117,A -85,B 0,C 180,E1 -8893.374,E2 -8893.374} C_VEL
LIN {X 0,Y 445.936,Z 560.317,A -85,B 0,C 180,E1 -8893.959,E2 -8893.959} C_VEL
LIN {X 0,Y 442.541,Z 568.11,A -85,B 0,C 180,E1 -8894.605,E2 -8894.605} C_VEL
LIN {X 0,Y 441.477,Z 572.611,A -85,B 0,C 180,E1 -8895.067,E2 -8895.067} C_VEL
LIN {X 0,Y 440.669,Z 583.113,A -85,B 0,C 180,E1 -8896.368,E2 -8896.368} C_VEL
LIN {X 0,Y 440.072,Z 592.504,A -85,B 0,C 180,E1 -8897.783,E2 -8897.783} C_VEL
LIN {X 0,Y 439.332,Z 601.265,A -85,B 0,C 180,E1 -8899.398,E2 -8899.398} C_VEL
LIN {X 0,Y 438.962,Z 607.453,A -85,B 0,C 180,E1 -8900.786,E2 -8900.786} C_VEL
LIN {X 0,Y 438.606,Z 613.994,A -85,B 0,C 180,E1 -8902.634,E2 -8902.634} C_VEL
LIN {X 0,Y 438.46,Z 618.898,A -85,B 0,C 180,E1 -8904.48,E2 -8904.48} C_VEL
LIN {X 0,Y 438.28,Z 622.32,A -85,B 0,C 180,E1 -8906.321,E2 -8906.321} C_VEL
LIN {X 0,Y 438.273,Z 624.357,A -85,B 0,C 180,E1 -8908.161,E2 -8908.161} C_VEL
LIN {X 0,Y 438.227,Z 625.063,A -85,B 0,C 180,E1 -8909.999,E2 -8909.999} C_VEL
LIN {X 0,Y 438.272,Z 624.438,A -85,B 0,C 180,E1 -8911.837,E2 -8911.837} C_VEL
LIN {X 0,Y 438.279,Z 622.469,A -85,B 0,C 180,E1 -8913.676,E2 -8913.676} C_VEL
LIN {X 0,Y 438.458,Z 619.114,A -85,B 0,C 180,E1 -8915.518,E2 -8915.518} C_VEL
LIN {X 0,Y 438.597,Z 614.276,A -85,B 0,C 180,E1 -8917.364,E2 -8917.364} C_VEL
LIN {X 0,Y 438.942,Z 607.813,A -85,B 0,C 180,E1 -8919.212,E2 -8919.212} C_VEL
LIN {X 0,Y 439.372,Z 600.609,A -85,B 0,C 180,E1 -8920.832,E2 -8920.832} C_VEL
LIN {X 0,Y 440.104,Z 591.639,A -85,B 0,C 180,E1 -8922.448,E2 -8922.448} C_VEL
LIN {X 0,Y 440.669,Z 582.256,A -85,B 0,C 180,E1 -8923.84,E2 -8923.84} C_VEL
LIN {X 0,Y 441.532,Z 571.867,A -85,B 0,C 180,E1 -8925.107,E2 -8925.107} C_VEL
LIN {X 0,Y 442.371,Z 560.41,A -85,B 0,C 180,E1 -8926.259,E2 -8926.259} C_VEL
LIN {X 0,Y 443.287,Z 547.718,A -85,B 0,C 180,E1 -8927.292,E2 -8927.292} C_VEL
LIN {X 0,Y 444.024,Z 534.618,A -85,B 0,C 180,E1 -8928.139,E2 -8928.139} C_VEL
LIN {X 0,Y 444.689,Z 520.198,A -85,B 0,C 180,E1 -8928.839,E2 -8928.839} C_VEL
LIN {X 0,Y 443.327,Z 511.602,A -85,B 0,C 180,E1 -8929.231,E2 -8929.231} C_VEL
LIN {X 0,Y 440.269,Z 498.143,A -85,B 0,C 180,E1 -8929.748,E2 -8929.748} C_VEL
LIN {X 0,Y 439.041,Z 492.91,A -85,B 0,C 180,E1 -8929.934,E2 -8929.934} C_VEL
LIN {X 0,Y 439.165,Z 486.16,A -85,B 0,C 180,E1 -8932.585,E2 -8932.585} C_VEL
LIN {X 0,Y 439.328,Z 478.773,A -85,B 0,C 180,E1 -8935.588,E2 -8935.588} C_VEL
LIN {X 0,Y 439.523,Z 471.412,A -85,B 0,C 180,E1 -8938.664,E2 -8938.664} C_VEL
LIN {X 0,Y 439.685,Z 465.282,A -85,B 0,C 180,E1 -8941.296,E2 -8941.296} C_VEL
LIN {X 0,Y 439.937,Z 457.664,A -85,B 0,C 180,E1 -8944.547,E2 -8944.547} C_VEL
LIN {X 0,Y 440.114,Z 449.721,A -85,B 0,C 180,E1 -8947.927,E2 -8947.927} C_VEL
LIN {X 0,Y 439.63,Z 445.199,A -85,B 0,C 180,E1 -8949.885,E2 -8949.885} C_VEL
LIN {X 0,Y 439.465,Z 444.372,A -85,B 0,C 180,E1 -8950.313,E2 -8950.313} C_VEL
LIN {X 0,Y 439.397,Z 444.378,A -85,B 0,C 180,E1 -8953.965,E2 -8953.965} C_VEL
LIN {X 0,Y 439.396,Z 444.379,A -85,B 0,C 180,E1 -8957.369,E2 -8957.369} C_VEL
LIN {X 0,Y 439.443,Z 444.369,A -85,B 0,C 180,E1 -8960.229,E2 -8960.229} C_VEL
LIN {X 0,Y 439.369,Z 444.38,A -85,B 0,C 180,E1 -8963.712,E2 -8963.712} C_VEL
LIN {X 0,Y 439.367,Z 444.382,A -85,B 0,C 180,E1 -8967.053,E2 -8967.053} C_VEL
LIN {X 0,Y 439.388,Z 444.38,A -85,B 0,C 180,E1 -8970.274,E2 -8970.274} C_VEL
LIN {X 0,Y 439.424,Z 444.37,A -85,B 0,C 180,E1 -8973.588,E2 -8973.588} C_VEL
LIN {X 0,Y 439.381,Z 444.378,A -85,B 0,C 180,E1 -8976.429,E2 -8976.429} C_VEL
LIN {X 0,Y 439.396,Z 444.373,A -85,B 0,C 180,E1 -8979.397,E2 -8979.397} C_VEL
LIN {X 0,Y 439.422,Z 444.375,A -85,B 0,C 180,E1 -8982.309,E2 -8982.309} C_VEL
LIN {X 0,Y 439.441,Z 444.37,A -85,B 0,C 180,E1 -8985.174,E2 -8985.174} C_VEL
LIN {X 0,Y 439.498,Z 444.36,A -85,B 0,C 180,E1 -8988.002,E2 -8988.002} C_VEL
LIN {X 0,Y 439.537,Z 444.355,A -85,B 0,C 180,E1 -8991.726,E2 -8991.726} C_VEL
LIN {X 0,Y 439.618,Z 444.347,A -85,B 0,C 180,E1 -8994.496,E2 -8994.496} C_VEL
LIN {X 0,Y 439.626,Z 444.345,A -85,B 0,C 180,E1 -8998.168,E2 -8998.168} C_VEL
LIN {X 0,Y 439.754,Z 444.331,A -85,B 0,C 180,E1 -9000,E2 -9000} C_VEL
LIN {X 0,Y 439.647,Z 444.337,A -85,B 0,C 180,E1 -9002.749,E2 -9002.749} C_VEL
LIN {X 0,Y 439.608,Z 444.352,A -85,B 0,C 180,E1 -9006.425,E2 -9006.425} C_VEL
LIN {X 0,Y 439.491,Z 444.36,A -85,B 0,C 180,E1 -9009.202,E2 -9009.202} C_VEL
LIN {X 0,Y 439.493,Z 444.36,A -85,B 0,C 180,E1 -9012.727,E2 -9012.727} C_VEL
LIN {X 0,Y 439.436,Z 444.368,A -85,B 0,C 180,E1 -9016.349,E2 -9016.349} C_VEL
LIN {X 0,Y 439.392,Z 444.374,A -85,B 0,C 180,E1 -9019.627,E2 -9019.627} C_VEL
LIN {X 0,Y 439.355,Z 444.38,A -85,B 0,C 180,E1 -9022.576,E2 -9022.576} C_VEL
LIN {X 0,Y 439.396,Z 444.378,A -85,B 0,C 180,E1 -9025.585,E2 -9025.585} C_VEL
LIN {X 0,Y 439.415,Z 444.374,A -85,B 0,C 180,E1 -9028.674,E2 -9028.674} C_VEL
LIN {X 0,Y 439.365,Z 444.379,A -85,B 0,C 180,E1 -9031.861,E2 -9031.861} C_VEL
LIN {X 0,Y 439.392,Z 444.377,A -85,B 0,C 180,E1 -9035.157,E2 -9035.157} C_VEL
LIN {X 0,Y 439.391,Z 444.376,A -85,B 0,C 180,E1 -9038.594,E2 -9038.594} C_VEL
LIN {X 0,Y 439.397,Z 444.377,A -85,B 0,C 180,E1 -9041.26,E2 -9041.26} C_VEL
LIN {X 0,Y 439.401,Z 444.378,A -85,B 0,C 180,E1 -9044.729,E2 -9044.729} C_VEL
LIN {X 0,Y 439.39,Z 444.38,A -85,B 0,C 180,E1 -9047.797,E2 -9047.797} C_VEL
LIN {X 0,Y 439.449,Z 444.455,A -85,B 0,C 180,E1 -9051.23,E2 -9051.23} C_VEL
LIN {X 0,Y 440.904,Z 452.386,A -85,B 0,C 180,E1 -9054.384,E2 -9054.384} C_VEL
LIN {X 0,Y 442.035,Z 458.559,A -85,B 0,C 180,E1 -9056.736,E2 -9056.736} C_VEL
LIN {X 0,Y 441.726,Z 464.524,A -85,B 0,C 180,E1 -9058.846,E2 -9058.846} C_VEL
LIN {X 0,Y 441.007,Z 473.6,A -85,B 0,C 180,E1 -9061.96,E2 -9061.96} C_VEL
LIN {X 0,Y 440.401,Z 482.671,A -85,B 0,C 180,E1 -9064.984,E2 -9064.984} C_VEL
LIN {X 0,Y 439.794,Z 493.264,A -85,B 0,C 180,E1 -9068.437,E2 -9068.437} C_VEL
LIN {X 0,Y 439.523,Z 499.385,A -85,B 0,C 180,E1 -9070.399,E2 -9070.399} C_VEL
LIN {X 0,Y 442.492,Z 514.693,A -85,B 0,C 180,E1 -9070.881,E2 -9070.881} C_VEL
LIN {X 0,Y 444.096,Z 526.31,A -85,B 0,C 180,E1 -9071.364,E2 -9071.364} C_VEL
LIN {X 0,Y 443.533,Z 540.022,A -85,B 0,C 180,E1 -9071.999,E2 -9071.999} C_VEL
LIN {X 0,Y 442.832,Z 553.189,A -85,B 0,C 180,E1 -9072.808,E2 -9072.808} C_VEL
LIN {X 0,Y 442.027,Z 565.04,A -85,B 0,C 180,E1 -9073.728,E2 -9073.728} C_VEL
LIN {X 0,Y 441.128,Z 577.028,A -85,B 0,C 180,E1 -9074.879,E2 -9074.879} C_VEL
LIN {X 0,Y 440.417,Z 587.82,A -85,B 0,C 180,E1 -9076.152,E2 -9076.152} C_VEL
LIN {X 0,Y 439.771,Z 597.645,A -85,B 0,C 180,E1 -9077.562,E2 -9077.562} C_VEL
LIN {X 0,Y 439.32,Z 605.543,A -85,B 0,C 180,E1 -9078.934,E2 -9078.934} C_VEL
LIN {X 0,Y 438.914,Z 612.205,A -85,B 0,C 180,E1 -9080.322,E2 -9080.322} C_VEL
LIN {X 0,Y 438.611,Z 617.724,A -85,B 0,C 180,E1 -9081.71,E2 -9081.71} C_VEL
LIN {X 0,Y 438.446,Z 623.496,A -85,B 0,C 180,E1 -9083.559,E2 -9083.559} C_VEL
LIN {X 0,Y 438.329,Z 627.686,A -85,B 0,C 180,E1 -9085.403,E2 -9085.403} C_VEL
LIN {X 0,Y 438.344,Z 630.419,A -85,B 0,C 180,E1 -9087.244,E2 -9087.244} C_VEL
LIN {X 0,Y 438.277,Z 631.773,A -85,B 0,C 180,E1 -9089.082,E2 -9089.082} C_VEL
LIN {X 0,Y 438.278,Z 631.772,A -85,B 0,C 180,E1 -9090.92,E2 -9090.92} C_VEL
LIN {X 0,Y 438.344,Z 630.412,A -85,B 0,C 180,E1 -9092.758,E2 -9092.758} C_VEL
LIN {X 0,Y 438.331,Z 627.675,A -85,B 0,C 180,E1 -9094.599,E2 -9094.599} C_VEL
LIN {X 0,Y 438.448,Z 623.487,A -85,B 0,C 180,E1 -9096.444,E2 -9096.444} C_VEL
LIN {X 0,Y 438.616,Z 617.713,A -85,B 0,C 180,E1 -9098.293,E2 -9098.293} C_VEL
LIN {X 0,Y 438.982,Z 611.181,A -85,B 0,C 180,E1 -9099.911,E2 -9099.911} C_VEL
LIN {X 0,Y 439.464,Z 603.046,A -85,B 0,C 180,E1 -9101.532,E2 -9101.532} C_VEL
LIN {X 0,Y 439.972,Z 594.024,A -85,B 0,C 180,E1 -9102.992,E2 -9102.992} C_VEL
LIN {X 0,Y 440.726,Z 584.114,A -85,B 0,C 180,E1 -9104.311,E2 -9104.311} C_VEL
LIN {X 0,Y 441.544,Z 572.47,A -85,B 0,C 180,E1 -9105.582,E2 -9105.582} C_VEL
LIN {X 0,Y 442.318,Z 560.785,A -85,B 0,C 180,E1 -9106.62,E2 -9106.62} C_VEL
LIN {X 0,Y 443.134,Z 547.882,A -85,B 0,C 180,E1 -9107.539,E2 -9107.539} C_VEL
LIN {X 0,Y 443.753,Z 535.282,A -85,B 0,C 180,E1 -9108.241,E2 -9108.241} C_VEL
LIN {X 0,Y 444.083,Z 525.192,A -85,B 0,C 180,E1 -9108.679,E2 -9108.679} C_VEL
LIN {X 0,Y 441.17,Z 506.374,A -85,B 0,C 180,E1 -9109.43,E2 -9109.43} C_VEL
LIN {X 0,Y 439.526,Z 498.722,A -85,B 0,C 180,E1 -9109.72,E2 -9109.72} C_VEL
LIN {X 0,Y 440.037,Z 488.783,A -85,B 0,C 180,E1 -9113.036,E2 -9113.036} C_VEL
LIN {X 0,Y 440.676,Z 480.379,A -85,B 0,C 180,E1 -9116.014,E2 -9116.014} C_VEL
LIN {X 0,Y 441.516,Z 472.804,A -85,B 0,C 180,E1 -9118.898,E2 -9118.898} C_VEL
LIN {X 0,Y 442.656,Z 465.16,A -85,B 0,C 180,E1 -9122.133,E2 -9122.133} C_VEL
LIN {X 0,Y 442.838,Z 461.863,A -85,B 0,C 180,E1 -9123.744,E2 -9123.744} C_VEL
LIN {X 0,Y 442.161,Z 458.053,A -85,B 0,C 180,E1 -9126.024,E2 -9126.024} C_VEL
LIN {X 0,Y 441.523,Z 454.443,A -85,B 0,C 180,E1 -9128.743,E2 -9128.743} C_VEL
LIN {X 0,Y 441.102,Z 452.472,A -85,B 0,C 180,E1 -9130.788,E2 -9130.788} C_VEL
LIN {X 0,Y 440.755,Z 450.961,A -85,B 0,C 180,E1 -9133.288,E2 -9133.288} C_VEL
LIN {X 0,Y 440.619,Z 450.414,A -85,B 0,C 180,E1 -9135.871,E2 -9135.871} C_VEL
LIN {X 0,Y 440.701,Z 450.87,A -85,B 0,C 180,E1 -9138.55,E2 -9138.55} C_VEL
LIN {X 0,Y 440.924,Z 452.503,A -85,B 0,C 180,E1 -9141.565,E2 -9141.565} C_VEL
LIN {X 0,Y 441.032,Z 454.435,A -85,B 0,C 180,E1 -9143.871,E2 -9143.871} C_VEL
LIN {X 0,Y 440.751,Z 456.815,A -85,B 0,C 180,E1 -9146.076,E2 -9146.076} C_VEL
LIN {X 0,Y 440.265,Z 460.87,A -85,B 0,C 180,E1 -9149.282,E2 -9149.282} C_VEL
LIN {X 0,Y 439.838,Z 465.273,A -85,B 0,C 180,E1 -9152.395,E2 -9152.395} C_VEL
LIN {X 0,Y 439.454,Z 470.375,A -85,B 0,C 180,E1 -9155.726,E2 -9155.726} C_VEL
LIN {X 0,Y 439.269,Z 474.699,A -85,B 0,C 180,E1 -9158.409,E2 -9158.409} C_VEL
LIN {X 0,Y 439.019,Z 479.601,A -85,B 0,C 180,E1 -9161.327,E2 -9161.327} C_VEL
LIN {X 0,Y 438.919,Z 482.658,A -85,B 0,C 180,E1 -9163.099,E2 -9163.099} C_VEL
LIN {X 0,Y 442.025,Z 494.396,A -85,B 0,C 180,E1 -9163.693,E2 -9163.693} C_VEL
LIN {X 0,Y 443.524,Z 502.853,A -85,B 0,C 180,E1 -9164.167,E2 -9164.167} C_VEL
LIN {X 0,Y 442.835,Z 516.247,A -85,B 0,C 180,E1 -9164.937,E2 -9164.937} C_VEL
LIN {X 0,Y 442.218,Z 527.05,A -85,B 0,C 180,E1 -9165.732,E2 -9165.732} C_VEL
LIN {X 0,Y 441.476,Z 538.411,A -85,B 0,C 180,E1 -9166.771,E2 -9166.771} C_VEL
LIN {X 0,Y 440.835,Z 547.726,A -85,B 0,C 180,E1 -9167.805,E2 -9167.805} C_VEL
LIN {X 0,Y 440.233,Z 556.326,A -85,B 0,C 180,E1 -9168.956,E2 -9168.956} C_VEL
LIN {X 0,Y 439.696,Z 564.786,A -85,B 0,C 180,E1 -9170.338,E2 -9170.338} C_VEL
LIN {X 0,Y 439.207,Z 571.589,A -85,B 0,C 180,E1 -9171.72,E2 -9171.72} C_VEL
LIN {X 0,Y 438.854,Z 577.287,A -85,B 0,C 180,E1 -9173.171,E2 -9173.171} C_VEL
LIN {X 0,Y 438.613,Z 581.339,A -85,B 0,C 180,E1 -9174.483,E2 -9174.483} C_VEL
LIN {X 0,Y 438.587,Z 583.608,A -85,B 0,C 180,E1 -9175.405,E2 -9175.405} C_VEL
LIN {X 0,Y 438.552,Z 585.444,A -85,B 0,C 180,E1 -9176.325,E2 -9176.325} C_VEL
LIN {X 0,Y 438.447,Z 586.815,A -85,B 0,C 180,E1 -9177.244,E2 -9177.244} C_VEL
LIN {X 0,Y 438.387,Z 587.775,A -85,B 0,C 180,E1 -9178.163,E2 -9178.163} C_VEL
LIN {X 0,Y 438.352,Z 588.341,A -85,B 0,C 180,E1 -9179.081,E2 -9179.081} C_VEL
LIN {X 0,Y 438.339,Z 588.51,A -85,B 0,C 180,E1 -9180,E2 -9180} C_VEL
